REGION Network 6: Safety control condition 3
   // Do not allow any motion when the Object is in a collision with axes.
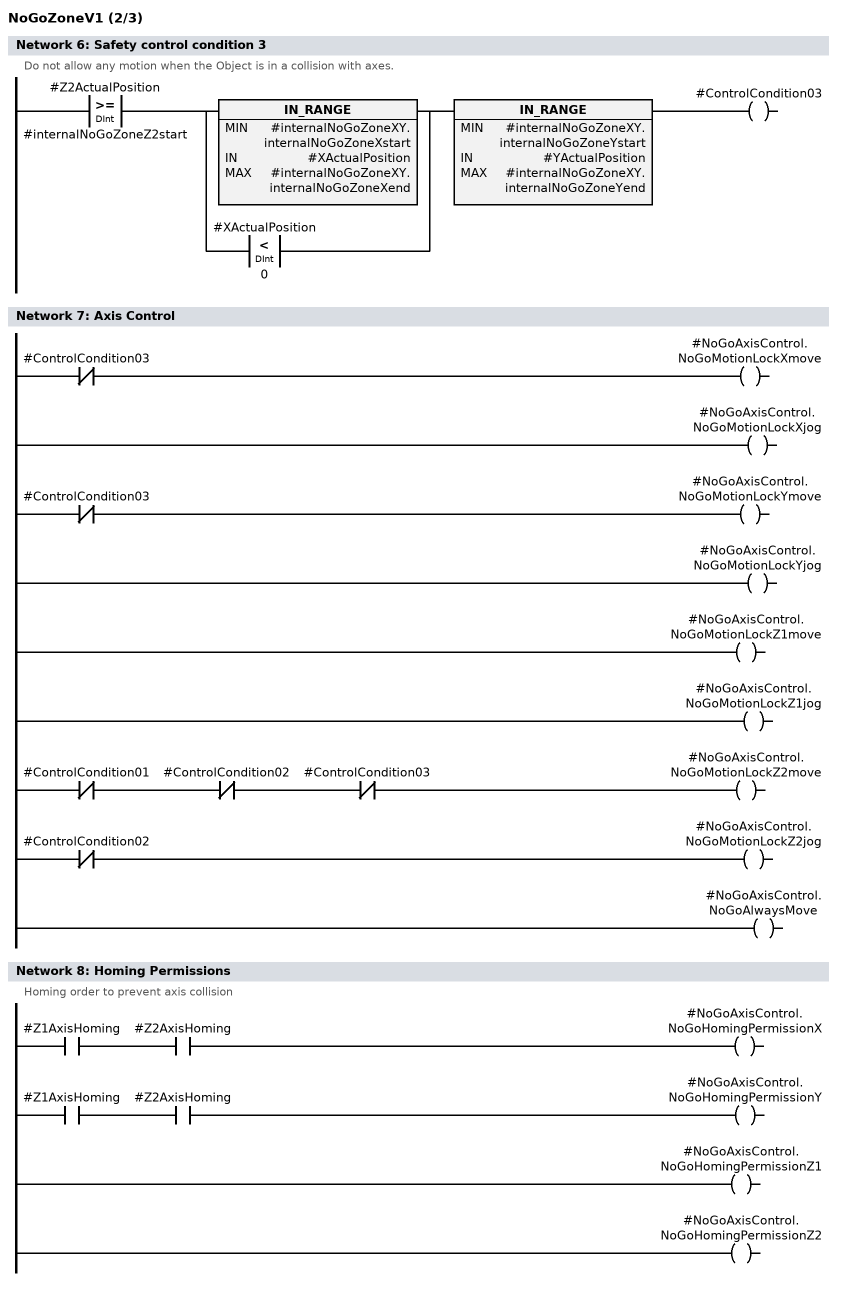
   RUNG wire#powerrail
      { S7_Templates := "SrcType := DInt" } GE_Contact(in1 := #Z2ActualPosition, in2 := #internalNoGoZoneZ2start)
      wire#w1
      { S7_Templates := "SrcType := DInt" } InRange(min := #internalNoGoZoneXY.internalNoGoZoneXstart, in := #XActualPosition, max := #internalNoGoZoneXY.internalNoGoZoneXend)
      wire#w2
      { S7_Templates := "SrcType := DInt" } InRange(min := #internalNoGoZoneXY.internalNoGoZoneYstart, in := #YActualPosition, max := #internalNoGoZoneXY.internalNoGoZoneYend)
      Coil( #ControlCondition03 )
   END_RUNG
   RUNG wire#w1
      { S7_Templates := "SrcType := DInt" } LT_Contact(in1 := #XActualPosition, in2 := 0)
   END_RUNG wire#w2
   // the same network as SCL:
   #ControlCondition03 := (#Z2ActualPosition >= #internalNoGoZoneZ2start) AND (((#internalNoGoZoneXY.internalNoGoZoneXstart <= #XActualPosition) AND (#XActualPosition <= #internalNoGoZoneXY.internalNoGoZoneXend)) OR (#XActualPosition < 0)) AND (#internalNoGoZoneXY.internalNoGoZoneYstart <= #YActualPosition) AND (#YActualPosition <= #internalNoGoZoneXY.internalNoGoZoneYend);
END_REGION

REGION Network 7: Axis Control
   RUNG wire#powerrail
      I_Contact( #ControlCondition03 )
      Coil( #NoGoAxisControl.NoGoMotionLockXmove )
   END_RUNG
   RUNG wire#powerrail
      Coil( #NoGoAxisControl.NoGoMotionLockXjog )
   END_RUNG
   RUNG wire#powerrail
      I_Contact( #ControlCondition03 )
      Coil( #NoGoAxisControl.NoGoMotionLockYmove )
   END_RUNG
   RUNG wire#powerrail
      Coil( #NoGoAxisControl.NoGoMotionLockYjog )
   END_RUNG
   RUNG wire#powerrail
      Coil( #NoGoAxisControl.NoGoMotionLockZ1move )
   END_RUNG
   RUNG wire#powerrail
      Coil( #NoGoAxisControl.NoGoMotionLockZ1jog )
   END_RUNG
   RUNG wire#powerrail
      I_Contact( #ControlCondition01 )
      I_Contact( #ControlCondition02 )
      I_Contact( #ControlCondition03 )
      Coil( #NoGoAxisControl.NoGoMotionLockZ2move )
   END_RUNG
   RUNG wire#powerrail
      I_Contact( #ControlCondition02 )
      Coil( #NoGoAxisControl.NoGoMotionLockZ2jog )
   END_RUNG
   RUNG wire#powerrail
      Coil( #NoGoAxisControl.NoGoAlwaysMove )
   END_RUNG
   // the same network as SCL:
   #NoGoAxisControl.NoGoMotionLockXmove := NOT #ControlCondition03;
   #NoGoAxisControl.NoGoMotionLockXjog := TRUE;
   #NoGoAxisControl.NoGoMotionLockYmove := NOT #ControlCondition03;
   #NoGoAxisControl.NoGoMotionLockYjog := TRUE;
   #NoGoAxisControl.NoGoMotionLockZ1move := TRUE;
   #NoGoAxisControl.NoGoMotionLockZ1jog := TRUE;
   #NoGoAxisControl.NoGoMotionLockZ2move := NOT #ControlCondition01 AND NOT #ControlCondition02 AND NOT #ControlCondition03;
   #NoGoAxisControl.NoGoMotionLockZ2jog := NOT #ControlCondition02;
   #NoGoAxisControl.NoGoAlwaysMove := TRUE;
END_REGION

REGION Network 8: Homing Permissions
   // Homing order to prevent axis collision
   RUNG wire#powerrail
      Contact( #Z1AxisHoming )
      Contact( #Z2AxisHoming )
      Coil( #NoGoAxisControl.NoGoHomingPermissionX )
   END_RUNG
   RUNG wire#powerrail
      Contact( #Z1AxisHoming )
      Contact( #Z2AxisHoming )
      Coil( #NoGoAxisControl.NoGoHomingPermissionY )
   END_RUNG
   RUNG wire#powerrail
      Coil( #NoGoAxisControl.NoGoHomingPermissionZ1 )
   END_RUNG
   RUNG wire#powerrail
      Coil( #NoGoAxisControl.NoGoHomingPermissionZ2 )
   END_RUNG
   // the same network as SCL:
   #NoGoAxisControl.NoGoHomingPermissionX := #Z1AxisHoming AND #Z2AxisHoming;
   #NoGoAxisControl.NoGoHomingPermissionY := #Z1AxisHoming AND #Z2AxisHoming;
   #NoGoAxisControl.NoGoHomingPermissionZ1 := TRUE;
   #NoGoAxisControl.NoGoHomingPermissionZ2 := TRUE;
END_REGION

REGION Network 9: Status
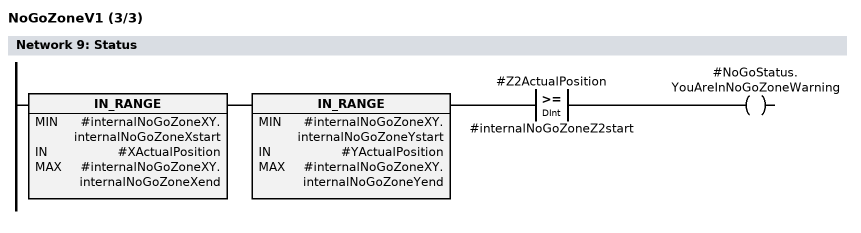
   RUNG wire#powerrail
      { S7_Templates := "SrcType := DInt" } InRange(min := #internalNoGoZoneXY.internalNoGoZoneXstart, in := #XActualPosition, max := #internalNoGoZoneXY.internalNoGoZoneXend)
      { S7_Templates := "SrcType := DInt" } InRange(min := #internalNoGoZoneXY.internalNoGoZoneYstart, in := #YActualPosition, max := #internalNoGoZoneXY.internalNoGoZoneYend)
      { S7_Templates := "SrcType := DInt" } GE_Contact(in1 := #Z2ActualPosition, in2 := #internalNoGoZoneZ2start)
      Coil( #NoGoStatus.YouAreInNoGoZoneWarning )
   END_RUNG
   // the same network as SCL:
   #NoGoStatus.YouAreInNoGoZoneWarning := (#internalNoGoZoneXY.internalNoGoZoneXstart <= #XActualPosition) AND (#XActualPosition <= #internalNoGoZoneXY.internalNoGoZoneXend) AND (#internalNoGoZoneXY.internalNoGoZoneYstart <= #YActualPosition) AND (#YActualPosition <= #internalNoGoZoneXY.internalNoGoZoneYend) AND (#Z2ActualPosition >= #internalNoGoZoneZ2start);
END_REGION
END_FUNCTION_BLOCK

FUNCTION "Reset Error" : Void   // FC15, LAD
{ S7_Optimized_Access := 'TRUE' }
AUTHOR : HenriP
VERSION : 0.1
   VAR_INPUT
      FestoAxisFault : Bool;
   END_VAR
   VAR_IN_OUT
      ResetCommand : Bool;
      FestoReset : Bool;
   END_VAR
BEGIN

REGION Network 1: Send Reset Command Flip Flop logic on Command
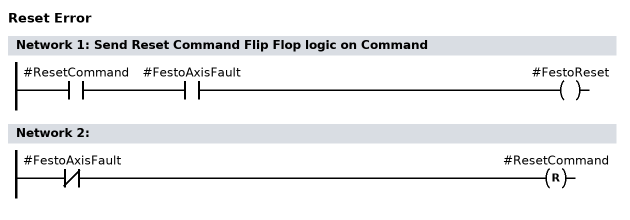
   RUNG wire#powerrail
      Contact( #ResetCommand )
      Contact( #FestoAxisFault )
      Coil( #FestoReset )
   END_RUNG
   // the same network as SCL:
   #FestoReset := #ResetCommand AND #FestoAxisFault;
END_REGION

REGION Network 2
   RUNG wire#powerrail
      I_Contact( #FestoAxisFault )
      R_Coil( #ResetCommand )
   END_RUNG
   // the same network as SCL:
   IF NOT #FestoAxisFault THEN #ResetCommand := FALSE; END_IF;
END_REGION
END_FUNCTION

ORGANIZATION_BLOCK "Startup"   // OB100, LAD, Startup
TITLE = "Complete Restart"
{ S7_Optimized_Access := 'TRUE' }
AUTHOR : HenriP
VERSION : 0.1
   VAR_INPUT
      LostRetentive : Bool;   // True if retentive data are lost
      LostRTC : Bool;   // True if date and time are lost
   END_VAR
   VAR_TEMP
      InitCall : Bool;
   END_VAR
BEGIN

REGION Network 1: Startup
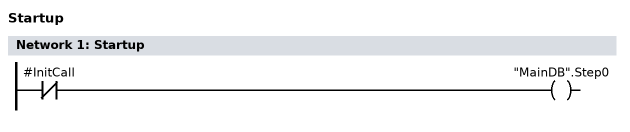
   RUNG wire#powerrail
      I_Contact( #InitCall )
      Coil( "MainDB".Step0 )
   END_RUNG
   // the same network as SCL:
   "MainDB".Step0 := NOT #InitCall;
END_REGION
END_ORGANIZATION_BLOCK

ORGANIZATION_BLOCK "Status Monitor"   // OB127, LAD, ProgramCycle
TITLE = Main Control block
{ S7_Optimized_Access := 'TRUE' }
AUTHOR : HenriP
VERSION : 0.1
   VAR_INPUT
      Initial_Call : Bool;   // Initial call of this OB
      Remanence : Bool;   // =True, if remanent data are available
   END_VAR
   VAR_TEMP
      ClearError : Bool;
   END_VAR
   VAR_TEMP   // added for the SCL form of the ladder/FBD networks
      _w1 : Bool;
   END_VAR
BEGIN

REGION Network 1: Monitor
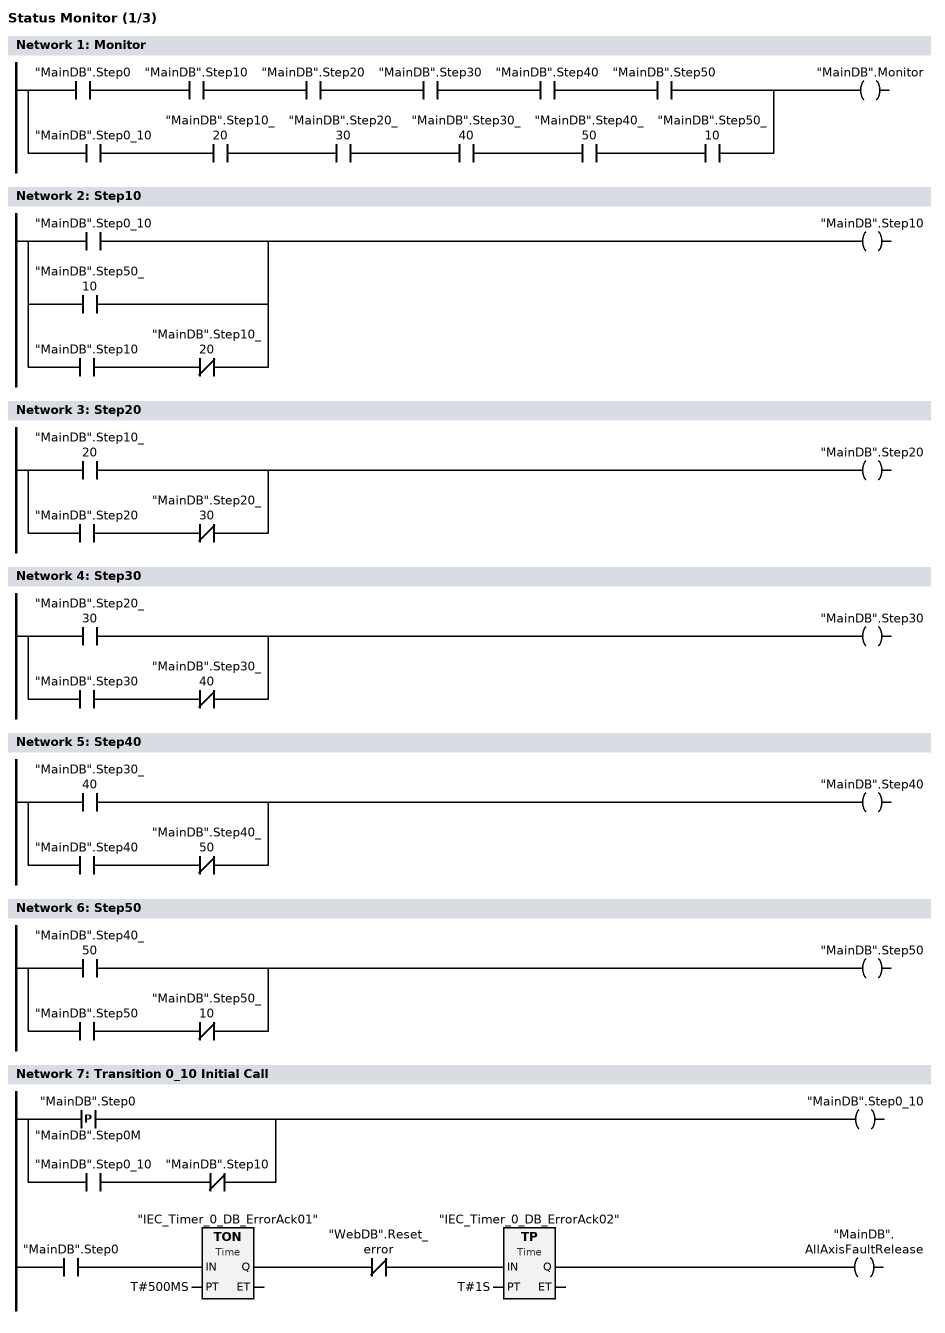
   RUNG wire#powerrail
      Contact( "MainDB".Step0 )
      Contact( "MainDB".Step10 )
      Contact( "MainDB".Step20 )
      Contact( "MainDB".Step30 )
      Contact( "MainDB".Step40 )
      Contact( "MainDB".Step50 )
      wire#w1
      Coil( "MainDB".Monitor )
   END_RUNG
   RUNG wire#powerrail
      Contact( "MainDB".Step0_10 )
      Contact( "MainDB".Step10_20 )
      Contact( "MainDB".Step20_30 )
      Contact( "MainDB".Step30_40 )
      Contact( "MainDB".Step40_50 )
      Contact( "MainDB".Step50_10 )
   END_RUNG wire#w1
   // the same network as SCL:
   "MainDB".Monitor := ("MainDB".Step0 AND "MainDB".Step10 AND "MainDB".Step20 AND "MainDB".Step30 AND "MainDB".Step40 AND "MainDB".Step50) OR ("MainDB".Step0_10 AND "MainDB".Step10_20 AND "MainDB".Step20_30 AND "MainDB".Step30_40 AND "MainDB".Step40_50 AND "MainDB".Step50_10);
END_REGION

REGION Network 2: Step10
   RUNG wire#powerrail
      Contact( "MainDB".Step0_10 )
      wire#w1
      Coil( "MainDB".Step10 )
   END_RUNG
   RUNG wire#powerrail
      Contact( "MainDB".Step50_10 )
   END_RUNG wire#w1
   RUNG wire#powerrail
      Contact( "MainDB".Step10 )
      I_Contact( "MainDB".Step10_20 )
   END_RUNG wire#w1
   // the same network as SCL:
   "MainDB".Step10 := "MainDB".Step0_10 OR "MainDB".Step50_10 OR ("MainDB".Step10 AND NOT "MainDB".Step10_20);
END_REGION

REGION Network 3: Step20
   RUNG wire#powerrail
      Contact( "MainDB".Step10_20 )
      wire#w1
      Coil( "MainDB".Step20 )
   END_RUNG
   RUNG wire#powerrail
      Contact( "MainDB".Step20 )
      I_Contact( "MainDB".Step20_30 )
   END_RUNG wire#w1
   // the same network as SCL:
   "MainDB".Step20 := "MainDB".Step10_20 OR ("MainDB".Step20 AND NOT "MainDB".Step20_30);
END_REGION

REGION Network 4: Step30
   RUNG wire#powerrail
      Contact( "MainDB".Step20_30 )
      wire#w1
      Coil( "MainDB".Step30 )
   END_RUNG
   RUNG wire#powerrail
      Contact( "MainDB".Step30 )
      I_Contact( "MainDB".Step30_40 )
   END_RUNG wire#w1
   // the same network as SCL:
   "MainDB".Step30 := "MainDB".Step20_30 OR ("MainDB".Step30 AND NOT "MainDB".Step30_40);
END_REGION

REGION Network 5: Step40
   RUNG wire#powerrail
      Contact( "MainDB".Step30_40 )
      wire#w1
      Coil( "MainDB".Step40 )
   END_RUNG
   RUNG wire#powerrail
      Contact( "MainDB".Step40 )
      I_Contact( "MainDB".Step40_50 )
   END_RUNG wire#w1
   // the same network as SCL:
   "MainDB".Step40 := "MainDB".Step30_40 OR ("MainDB".Step40 AND NOT "MainDB".Step40_50);
END_REGION

REGION Network 6: Step50
   RUNG wire#powerrail
      Contact( "MainDB".Step40_50 )
      wire#w1
      Coil( "MainDB".Step50 )
   END_RUNG
   RUNG wire#powerrail
      Contact( "MainDB".Step50 )
      I_Contact( "MainDB".Step50_10 )
   END_RUNG wire#w1
   // the same network as SCL:
   "MainDB".Step50 := "MainDB".Step40_50 OR ("MainDB".Step50 AND NOT "MainDB".Step50_10);
END_REGION

REGION Network 7: Transition 0_10 Initial Call
   RUNG wire#powerrail
      P_Contact(operand := "MainDB".Step0, bit := "MainDB".Step0M)
      wire#w1
      Coil( "MainDB".Step0_10 )
   END_RUNG
   RUNG wire#powerrail
      Contact( "MainDB".Step0_10 )
      I_Contact( "MainDB".Step10 )
   END_RUNG wire#w1
   RUNG wire#powerrail
      Contact( "MainDB".Step0 )
      { S7_Templates := "time_type := Time" } "IEC_Timer_0_DB_ErrorAck01".TON(pt := T#500MS, et =>)
      I_Contact( "WebDB".Reset_error )
      { S7_Templates := "time_type := Time" } "IEC_Timer_0_DB_ErrorAck02".TP(pt := T#1S, et =>)
      Coil( "MainDB".AllAxisFaultRelease )
   END_RUNG
   // the same network as SCL:
   #_w1 := "MainDB".Step0 AND NOT "MainDB".Step0M;   // rising edge of "MainDB".Step0
   "MainDB".Step0M := "MainDB".Step0;
   "MainDB".Step0_10 := #_w1 OR ("MainDB".Step0_10 AND NOT "MainDB".Step10);
   "IEC_Timer_0_DB_ErrorAck01".TON(IN := "MainDB".Step0, PT := T#500MS);
   "IEC_Timer_0_DB_ErrorAck02".TP(IN := "IEC_Timer_0_DB_ErrorAck01".Q AND NOT "WebDB".Reset_error, PT := T#1S);
   "MainDB".AllAxisFaultRelease := "IEC_Timer_0_DB_ErrorAck02".Q;
END_REGION

REGION Network 8: Transition10-20 Check PLC Operating State -> Wait Ready
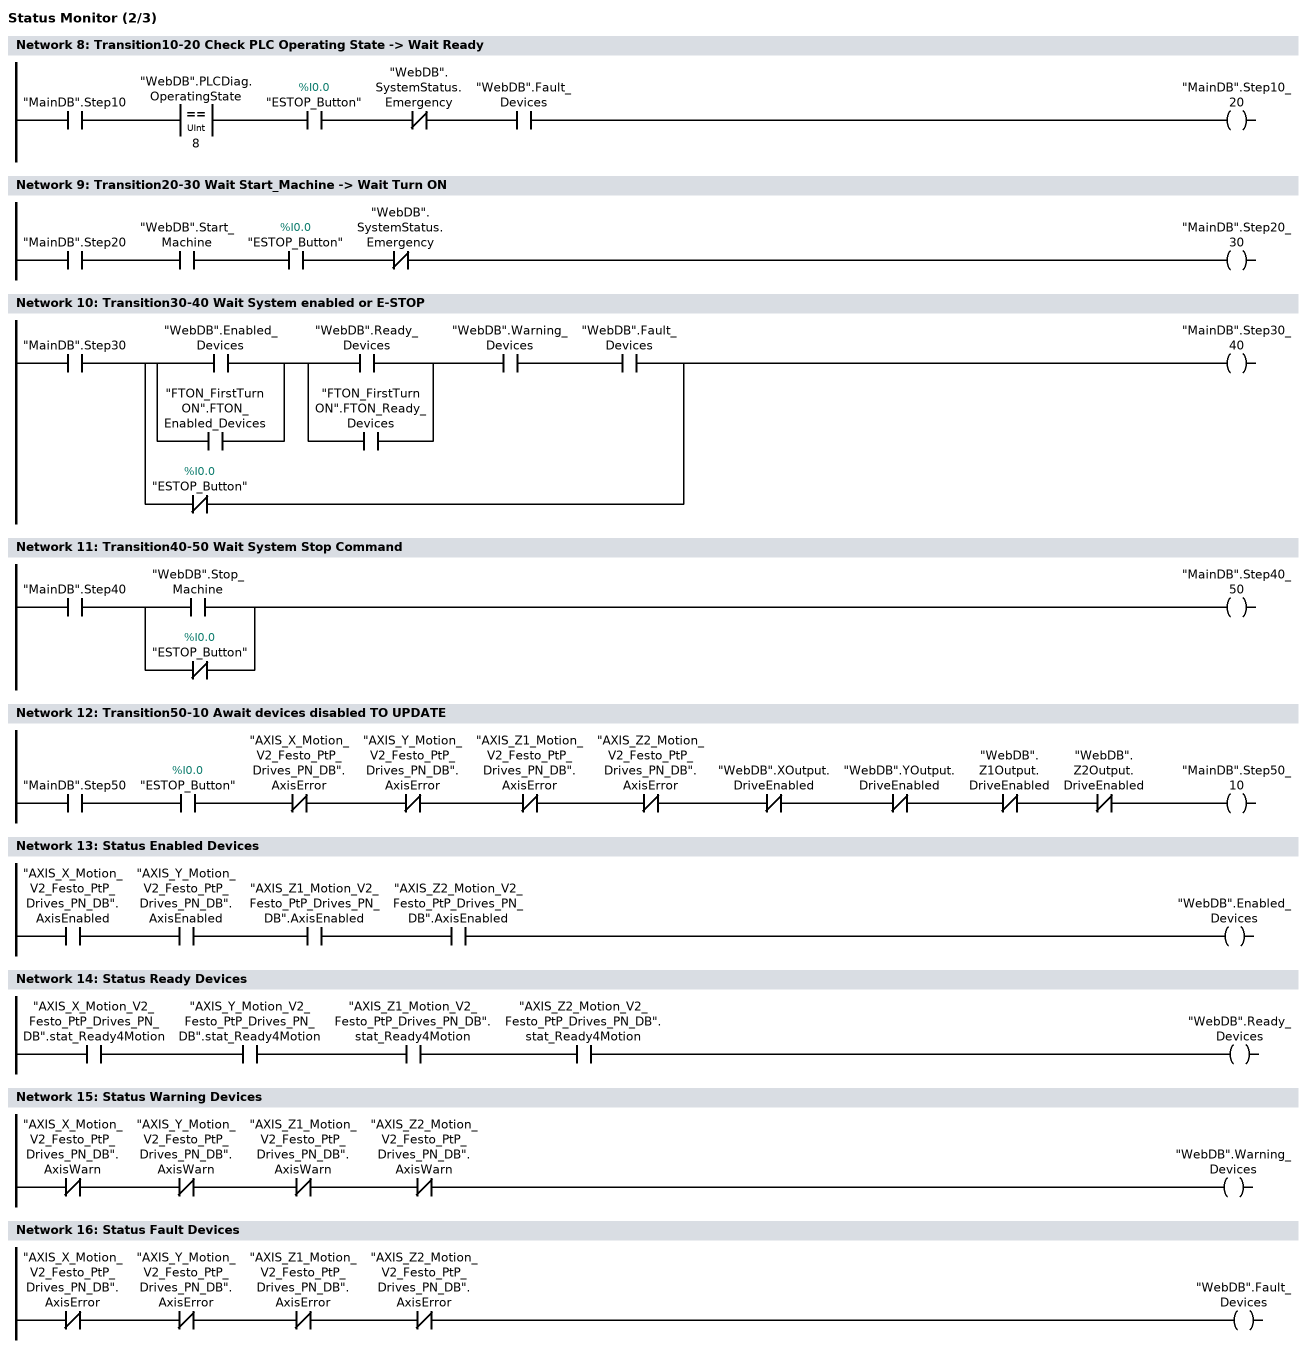
   RUNG wire#powerrail
      Contact( "MainDB".Step10 )
      { S7_Templates := "SrcType := UInt" } EQ_Contact(in1 := "WebDB".PLCDiag.OperatingState, in2 := 8)
      Contact( "ESTOP_Button" )
      I_Contact( "WebDB".SystemStatus.Emergency )
      Contact( "WebDB".Fault_Devices )
      Coil( "MainDB".Step10_20 )
   END_RUNG
   // the same network as SCL:
   "MainDB".Step10_20 := "MainDB".Step10 AND ("WebDB".PLCDiag.OperatingState = 8) AND "ESTOP_Button" AND NOT "WebDB".SystemStatus.Emergency AND "WebDB".Fault_Devices;
END_REGION

REGION Network 9: Transition20-30 Wait Start_Machine -> Wait Turn ON
   RUNG wire#powerrail
      Contact( "MainDB".Step20 )
      Contact( "WebDB".Start_Machine )
      Contact( "ESTOP_Button" )
      I_Contact( "WebDB".SystemStatus.Emergency )
      Coil( "MainDB".Step20_30 )
   END_RUNG
   // the same network as SCL:
   "MainDB".Step20_30 := "MainDB".Step20 AND "WebDB".Start_Machine AND "ESTOP_Button" AND NOT "WebDB".SystemStatus.Emergency;
END_REGION

REGION Network 10: Transition30-40 Wait System enabled or E-STOP
   RUNG wire#powerrail
      Contact( "MainDB".Step30 )
      wire#w1
      Contact( "WebDB".Enabled_Devices )
      wire#w2
      Contact( "WebDB".Ready_Devices )
      wire#w3
      Contact( "WebDB".Warning_Devices )
      Contact( "WebDB".Fault_Devices )
      wire#w4
      Coil( "MainDB".Step30_40 )
   END_RUNG
   RUNG wire#w1
      Contact( "FTON_FirstTurnON".FTON_Enabled_Devices )
   END_RUNG wire#w2
   RUNG wire#w2
      Contact( "FTON_FirstTurnON".FTON_Ready_Devices )
   END_RUNG wire#w3
   RUNG wire#w1
      I_Contact( "ESTOP_Button" )
   END_RUNG wire#w4
   // the same network as SCL:
   "MainDB".Step30_40 := "MainDB".Step30 AND ((("WebDB".Enabled_Devices OR "FTON_FirstTurnON".FTON_Enabled_Devices) AND ("WebDB".Ready_Devices OR "FTON_FirstTurnON".FTON_Ready_Devices) AND "WebDB".Warning_Devices AND "WebDB".Fault_Devices) OR NOT "ESTOP_Button");
END_REGION

REGION Network 11: Transition40-50 Wait System Stop Command
   RUNG wire#powerrail
      Contact( "MainDB".Step40 )
      wire#w1
      Contact( "WebDB".Stop_Machine )
      wire#w2
      Coil( "MainDB".Step40_50 )
   END_RUNG
   RUNG wire#w1
      I_Contact( "ESTOP_Button" )
   END_RUNG wire#w2
   // the same network as SCL:
   "MainDB".Step40_50 := "MainDB".Step40 AND ("WebDB".Stop_Machine OR NOT "ESTOP_Button");
END_REGION

REGION Network 12: Transition50-10 Await devices disabled TO UPDATE
   RUNG wire#powerrail
      Contact( "MainDB".Step50 )
      Contact( "ESTOP_Button" )
      I_Contact( "AXIS_X_Motion_V2_Festo_PtP_Drives_PN_DB".AxisError )
      I_Contact( "AXIS_Y_Motion_V2_Festo_PtP_Drives_PN_DB".AxisError )
      I_Contact( "AXIS_Z1_Motion_V2_Festo_PtP_Drives_PN_DB".AxisError )
      I_Contact( "AXIS_Z2_Motion_V2_Festo_PtP_Drives_PN_DB".AxisError )
      I_Contact( "WebDB".XOutput.DriveEnabled )
      I_Contact( "WebDB".YOutput.DriveEnabled )
      I_Contact( "WebDB".Z1Output.DriveEnabled )
      I_Contact( "WebDB".Z2Output.DriveEnabled )
      Coil( "MainDB".Step50_10 )
   END_RUNG
   // the same network as SCL:
   "MainDB".Step50_10 := "MainDB".Step50 AND "ESTOP_Button" AND NOT "AXIS_X_Motion_V2_Festo_PtP_Drives_PN_DB".AxisError AND NOT "AXIS_Y_Motion_V2_Festo_PtP_Drives_PN_DB".AxisError AND NOT "AXIS_Z1_Motion_V2_Festo_PtP_Drives_PN_DB".AxisError AND NOT "AXIS_Z2_Motion_V2_Festo_PtP_Drives_PN_DB".AxisError AND NOT "WebDB".XOutput.DriveEnabled AND NOT "WebDB".YOutput.DriveEnabled AND NOT "WebDB".Z1Output.DriveEnabled AND NOT "WebDB".Z2Output.DriveEnabled;
END_REGION

REGION Network 13: Status Enabled Devices
   RUNG wire#powerrail
      Contact( "AXIS_X_Motion_V2_Festo_PtP_Drives_PN_DB".AxisEnabled )
      Contact( "AXIS_Y_Motion_V2_Festo_PtP_Drives_PN_DB".AxisEnabled )
      Contact( "AXIS_Z1_Motion_V2_Festo_PtP_Drives_PN_DB".AxisEnabled )
      Contact( "AXIS_Z2_Motion_V2_Festo_PtP_Drives_PN_DB".AxisEnabled )
      Coil( "WebDB".Enabled_Devices )
   END_RUNG
   // the same network as SCL:
   "WebDB".Enabled_Devices := "AXIS_X_Motion_V2_Festo_PtP_Drives_PN_DB".AxisEnabled AND "AXIS_Y_Motion_V2_Festo_PtP_Drives_PN_DB".AxisEnabled AND "AXIS_Z1_Motion_V2_Festo_PtP_Drives_PN_DB".AxisEnabled AND "AXIS_Z2_Motion_V2_Festo_PtP_Drives_PN_DB".AxisEnabled;
END_REGION

REGION Network 14: Status Ready Devices
   RUNG wire#powerrail
      Contact( "AXIS_X_Motion_V2_Festo_PtP_Drives_PN_DB".stat_Ready4Motion )
      Contact( "AXIS_Y_Motion_V2_Festo_PtP_Drives_PN_DB".stat_Ready4Motion )
      Contact( "AXIS_Z1_Motion_V2_Festo_PtP_Drives_PN_DB".stat_Ready4Motion )
      Contact( "AXIS_Z2_Motion_V2_Festo_PtP_Drives_PN_DB".stat_Ready4Motion )
      Coil( "WebDB".Ready_Devices )
   END_RUNG
   // the same network as SCL:
   "WebDB".Ready_Devices := "AXIS_X_Motion_V2_Festo_PtP_Drives_PN_DB".stat_Ready4Motion AND "AXIS_Y_Motion_V2_Festo_PtP_Drives_PN_DB".stat_Ready4Motion AND "AXIS_Z1_Motion_V2_Festo_PtP_Drives_PN_DB".stat_Ready4Motion AND "AXIS_Z2_Motion_V2_Festo_PtP_Drives_PN_DB".stat_Ready4Motion;
END_REGION

REGION Network 15: Status Warning Devices
   RUNG wire#powerrail
      I_Contact( "AXIS_X_Motion_V2_Festo_PtP_Drives_PN_DB".AxisWarn )
      I_Contact( "AXIS_Y_Motion_V2_Festo_PtP_Drives_PN_DB".AxisWarn )
      I_Contact( "AXIS_Z1_Motion_V2_Festo_PtP_Drives_PN_DB".AxisWarn )
      I_Contact( "AXIS_Z2_Motion_V2_Festo_PtP_Drives_PN_DB".AxisWarn )
      Coil( "WebDB".Warning_Devices )
   END_RUNG
   // the same network as SCL:
   "WebDB".Warning_Devices := NOT "AXIS_X_Motion_V2_Festo_PtP_Drives_PN_DB".AxisWarn AND NOT "AXIS_Y_Motion_V2_Festo_PtP_Drives_PN_DB".AxisWarn AND NOT "AXIS_Z1_Motion_V2_Festo_PtP_Drives_PN_DB".AxisWarn AND NOT "AXIS_Z2_Motion_V2_Festo_PtP_Drives_PN_DB".AxisWarn;
END_REGION

REGION Network 16: Status Fault Devices
   RUNG wire#powerrail
      I_Contact( "AXIS_X_Motion_V2_Festo_PtP_Drives_PN_DB".AxisError )
      I_Contact( "AXIS_Y_Motion_V2_Festo_PtP_Drives_PN_DB".AxisError )
      I_Contact( "AXIS_Z1_Motion_V2_Festo_PtP_Drives_PN_DB".AxisError )
      I_Contact( "AXIS_Z2_Motion_V2_Festo_PtP_Drives_PN_DB".AxisError )
      Coil( "WebDB".Fault_Devices )
   END_RUNG
   // the same network as SCL:
   "WebDB".Fault_Devices := NOT "AXIS_X_Motion_V2_Festo_PtP_Drives_PN_DB".AxisError AND NOT "AXIS_Y_Motion_V2_Festo_PtP_Drives_PN_DB".AxisError AND NOT "AXIS_Z1_Motion_V2_Festo_PtP_Drives_PN_DB".AxisError AND NOT "AXIS_Z2_Motion_V2_Festo_PtP_Drives_PN_DB".AxisError;
END_REGION

REGION Network 17: Emergency button is active
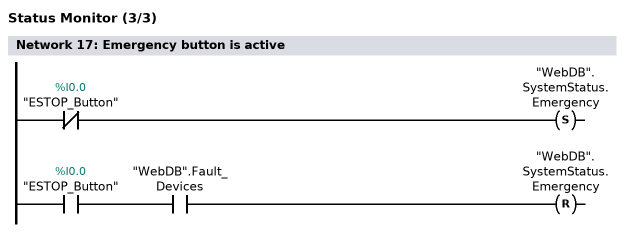
   RUNG wire#powerrail
      I_Contact( "ESTOP_Button" )
      S_Coil( "WebDB".SystemStatus.Emergency )
   END_RUNG
   RUNG wire#powerrail
      Contact( "ESTOP_Button" )
      Contact( "WebDB".Fault_Devices )
      R_Coil( "WebDB".SystemStatus.Emergency )
   END_RUNG
   // the same network as SCL:
   IF NOT "ESTOP_Button" THEN "WebDB".SystemStatus.Emergency := TRUE; END_IF;
   IF "ESTOP_Button" AND "WebDB".Fault_Devices THEN "WebDB".SystemStatus.Emergency := FALSE; END_IF;
END_REGION
END_ORGANIZATION_BLOCK

ORGANIZATION_BLOCK "Work"   // OB123, LAD, ProgramCycle
TITLE = "Main Program Sweep (Cycle)"
{ S7_Optimized_Access := 'TRUE' }
VERSION : 0.1
   VAR_INPUT
      Initial_Call : Bool;   // Initial call of this OB
      Remanence : Bool;   // =True, if remanent data are available
   END_VAR
BEGIN

REGION Network 1: Active machine
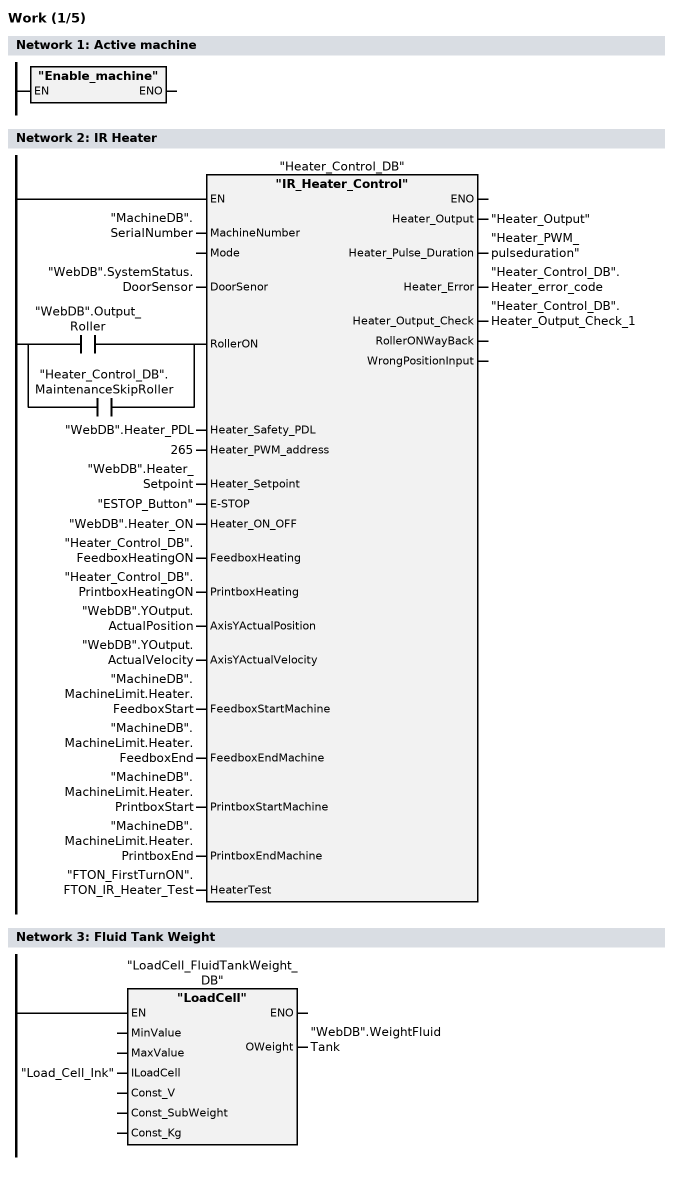
   RUNG wire#powerrail
      "Enable_machine"()
   END_RUNG
   // the same network as SCL:
   "Enable_machine"();
END_REGION

REGION Network 2: IR Heater
   RUNG wire#powerrail
      "Heater_Control_DB"(RollerON := wire#w1, MachineNumber := "MachineDB".SerialNumber, Mode :=, DoorSenor := "WebDB".SystemStatus.DoorSensor, Heater_Safety_PDL := "WebDB".Heater_PDL, Heater_PWM_address := 265, Heater_Setpoint := "WebDB".Heater_Setpoint, "E-STOP" := "ESTOP_Button", Heater_ON_OFF := "WebDB".Heater_ON, FeedboxHeating := "Heater_Control_DB".FeedboxHeatingON, PrintboxHeating := "Heater_Control_DB".PrintboxHeatingON, AxisYActualPosition := "WebDB".YOutput.ActualPosition, AxisYActualVelocity := "WebDB".YOutput.ActualVelocity, FeedboxStartMachine := "MachineDB".MachineLimit.Heater.FeedboxStart, FeedboxEndMachine := "MachineDB".MachineLimit.Heater.FeedboxEnd, PrintboxStartMachine := "MachineDB".MachineLimit.Heater.PrintboxStart, PrintboxEndMachine := "MachineDB".MachineLimit.Heater.PrintboxEnd, HeaterTest := "FTON_FirstTurnON".FTON_IR_Heater_Test, Heater_Output => "Heater_Output", Heater_Pulse_Duration => "Heater_PWM_pulseduration", Heater_Error => "Heater_Control_DB".Heater_error_code, Heater_Output_Check => "Heater_Control_DB".Heater_Output_Check_1, RollerONWayBack =>, WrongPositionInput =>)
   END_RUNG
   RUNG wire#powerrail
      Contact( "WebDB".Output_Roller )
   END_RUNG wire#w1
   RUNG wire#powerrail
      Contact( "Heater_Control_DB".MaintenanceSkipRoller )
   END_RUNG wire#w1
   // the same network as SCL:
   "Heater_Control_DB"(MachineNumber := "MachineDB".SerialNumber,   // "IR_Heater_Control"
                       DoorSenor := "WebDB".SystemStatus.DoorSensor,
                       RollerON := "WebDB".Output_Roller OR "Heater_Control_DB".MaintenanceSkipRoller,
                       Heater_Safety_PDL := "WebDB".Heater_PDL,
                       Heater_PWM_address := 265,
                       Heater_Setpoint := "WebDB".Heater_Setpoint,
                       "E-STOP" := "ESTOP_Button",
                       Heater_ON_OFF := "WebDB".Heater_ON,
                       FeedboxHeating := "Heater_Control_DB".FeedboxHeatingON,
                       PrintboxHeating := "Heater_Control_DB".PrintboxHeatingON,
                       AxisYActualPosition := "WebDB".YOutput.ActualPosition,
                       AxisYActualVelocity := "WebDB".YOutput.ActualVelocity,
                       FeedboxStartMachine := "MachineDB".MachineLimit.Heater.FeedboxStart,
                       FeedboxEndMachine := "MachineDB".MachineLimit.Heater.FeedboxEnd,
                       PrintboxStartMachine := "MachineDB".MachineLimit.Heater.PrintboxStart,
                       PrintboxEndMachine := "MachineDB".MachineLimit.Heater.PrintboxEnd,
                       HeaterTest := "FTON_FirstTurnON".FTON_IR_Heater_Test,
                       Heater_Output => "Heater_Output",
                       Heater_Pulse_Duration => "Heater_PWM_pulseduration",
                       Heater_Error => "Heater_Control_DB".Heater_error_code,
                       Heater_Output_Check => "Heater_Control_DB".Heater_Output_Check_1);
END_REGION

REGION Network 3: Fluid Tank Weight
   RUNG wire#powerrail
      "LoadCell_FluidTankWeight_DB"(MinValue :=, MaxValue :=, ILoadCell := "Load_Cell_Ink", Const_V :=, Const_SubWeight :=, Const_Kg :=, OWeight => "WebDB".WeightFluidTank)
   END_RUNG
   // the same network as SCL:
   "LoadCell_FluidTankWeight_DB"(ILoadCell := "Load_Cell_Ink", OWeight => "WebDB".WeightFluidTank);   // "LoadCell"
END_REGION

REGION Network 4: Fluid Waste Weight
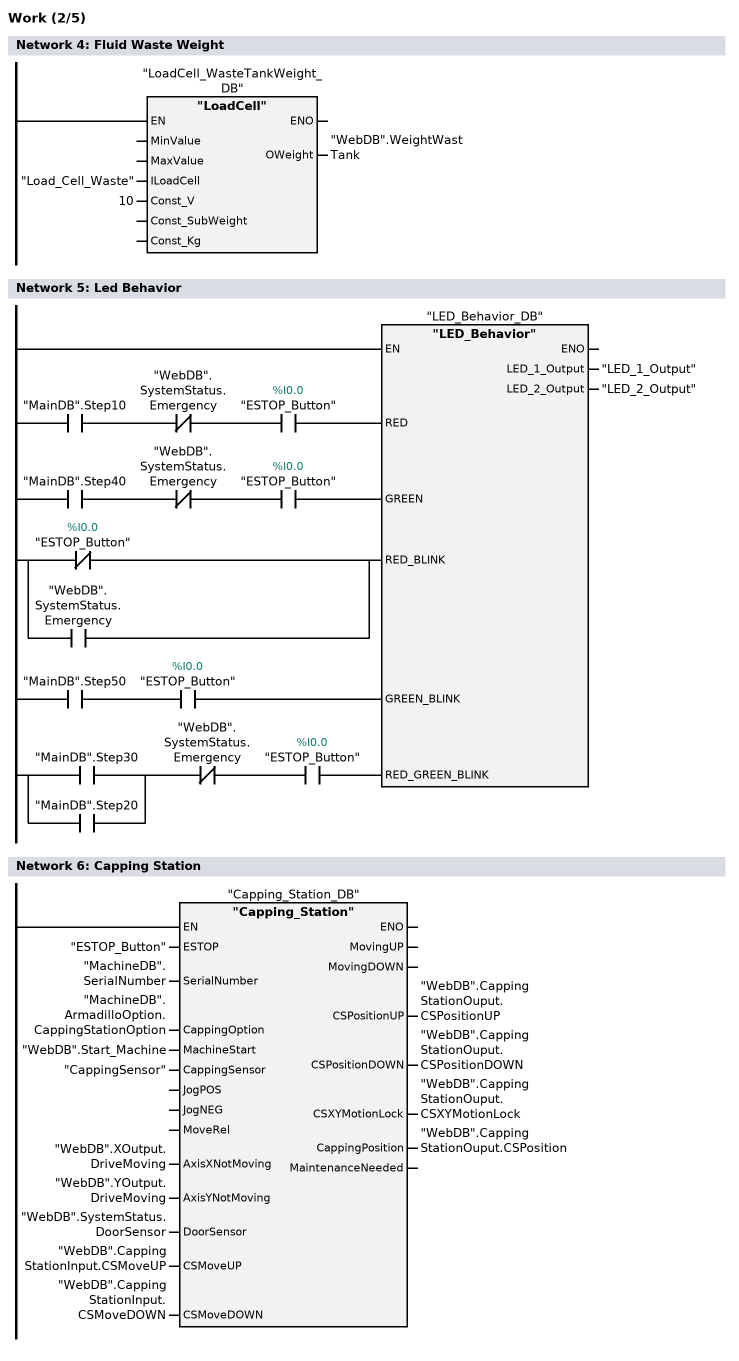
   RUNG wire#powerrail
      "LoadCell_WasteTankWeight_DB"(MinValue :=, MaxValue :=, ILoadCell := "Load_Cell_Waste", Const_V := 10, Const_SubWeight :=, Const_Kg :=, OWeight => "WebDB".WeightWastTank)
   END_RUNG
   // the same network as SCL:
   "LoadCell_WasteTankWeight_DB"(ILoadCell := "Load_Cell_Waste",   // "LoadCell"
                           Const_V := 10,
                           OWeight => "WebDB".WeightWastTank);
END_REGION

REGION Network 5: Led Behavior
   RUNG wire#powerrail
      "LED_Behavior_DB"(RED := wire#w1, GREEN := wire#w2, RED_BLINK := wire#w3, GREEN_BLINK := wire#w4, RED_GREEN_BLINK := wire#w6, LED_1_Output => "LED_1_Output", LED_2_Output => "LED_2_Output")
   END_RUNG
   RUNG wire#powerrail
      Contact( "MainDB".Step10 )
      I_Contact( "WebDB".SystemStatus.Emergency )
      Contact( "ESTOP_Button" )
   END_RUNG wire#w1
   RUNG wire#powerrail
      Contact( "MainDB".Step40 )
      I_Contact( "WebDB".SystemStatus.Emergency )
      Contact( "ESTOP_Button" )
   END_RUNG wire#w2
   RUNG wire#powerrail
      I_Contact( "ESTOP_Button" )
   END_RUNG wire#w3
   RUNG wire#powerrail
      Contact( "WebDB".SystemStatus.Emergency )
   END_RUNG wire#w3
   RUNG wire#powerrail
      Contact( "MainDB".Step50 )
      Contact( "ESTOP_Button" )
   END_RUNG wire#w4
   RUNG wire#powerrail
      Contact( "MainDB".Step30 )
      wire#w5
      I_Contact( "WebDB".SystemStatus.Emergency )
      Contact( "ESTOP_Button" )
   END_RUNG wire#w6
   RUNG wire#powerrail
      Contact( "MainDB".Step20 )
   END_RUNG wire#w5
   // the same network as SCL:
   "LED_Behavior_DB"(RED := "MainDB".Step10 AND NOT "WebDB".SystemStatus.Emergency AND "ESTOP_Button",   // "LED_Behavior"
                     GREEN := "MainDB".Step40 AND NOT "WebDB".SystemStatus.Emergency AND "ESTOP_Button",
                     RED_BLINK := NOT "ESTOP_Button" OR "WebDB".SystemStatus.Emergency,
                     GREEN_BLINK := "MainDB".Step50 AND "ESTOP_Button",
                     RED_GREEN_BLINK := ("MainDB".Step30 OR "MainDB".Step20) AND NOT "WebDB".SystemStatus.Emergency AND "ESTOP_Button",
                     LED_1_Output => "LED_1_Output",
                     LED_2_Output => "LED_2_Output");
END_REGION

REGION Network 6: Capping Station
   RUNG wire#powerrail
      "Capping_Station_DB"(ESTOP := "ESTOP_Button", SerialNumber := "MachineDB".SerialNumber, CappingOption := "MachineDB".ArmadilloOption.CappingStationOption, MachineStart := "WebDB".Start_Machine, CappingSensor := "CappingSensor", JogPOS :=, JogNEG :=, MoveRel :=, AxisXNotMoving := "WebDB".XOutput.DriveMoving, AxisYNotMoving := "WebDB".YOutput.DriveMoving, DoorSensor := "WebDB".SystemStatus.DoorSensor, CSMoveUP := "WebDB".CappingStationInput.CSMoveUP, CSMoveDOWN := "WebDB".CappingStationInput.CSMoveDOWN, MovingUP =>, MovingDOWN =>, CSPositionUP => "WebDB".CappingStationOuput.CSPositionUP, CSPositionDOWN => "WebDB".CappingStationOuput.CSPositionDOWN, CSXYMotionLock => "WebDB".CappingStationOuput.CSXYMotionLock, CappingPosition => "WebDB".CappingStationOuput.CSPosition, MaintenanceNeeded =>)
   END_RUNG
   // the same network as SCL:
   "Capping_Station_DB"(ESTOP := "ESTOP_Button",   // "Capping_Station"
                        SerialNumber := "MachineDB".SerialNumber,
                        CappingOption := "MachineDB".ArmadilloOption.CappingStationOption,
                        MachineStart := "WebDB".Start_Machine,
                        CappingSensor := "CappingSensor",
                        AxisXNotMoving := "WebDB".XOutput.DriveMoving,
                        AxisYNotMoving := "WebDB".YOutput.DriveMoving,
                        DoorSensor := "WebDB".SystemStatus.DoorSensor,
                        CSMoveUP := "WebDB".CappingStationInput.CSMoveUP,
                        CSMoveDOWN := "WebDB".CappingStationInput.CSMoveDOWN,
                        CSPositionUP => "WebDB".CappingStationOuput.CSPositionUP,
                        CSPositionDOWN => "WebDB".CappingStationOuput.CSPositionDOWN,
                        CSXYMotionLock => "WebDB".CappingStationOuput.CSXYMotionLock,
                        CappingPosition => "WebDB".CappingStationOuput.CSPosition);
END_REGION

REGION Network 7: Initial Test Sequence
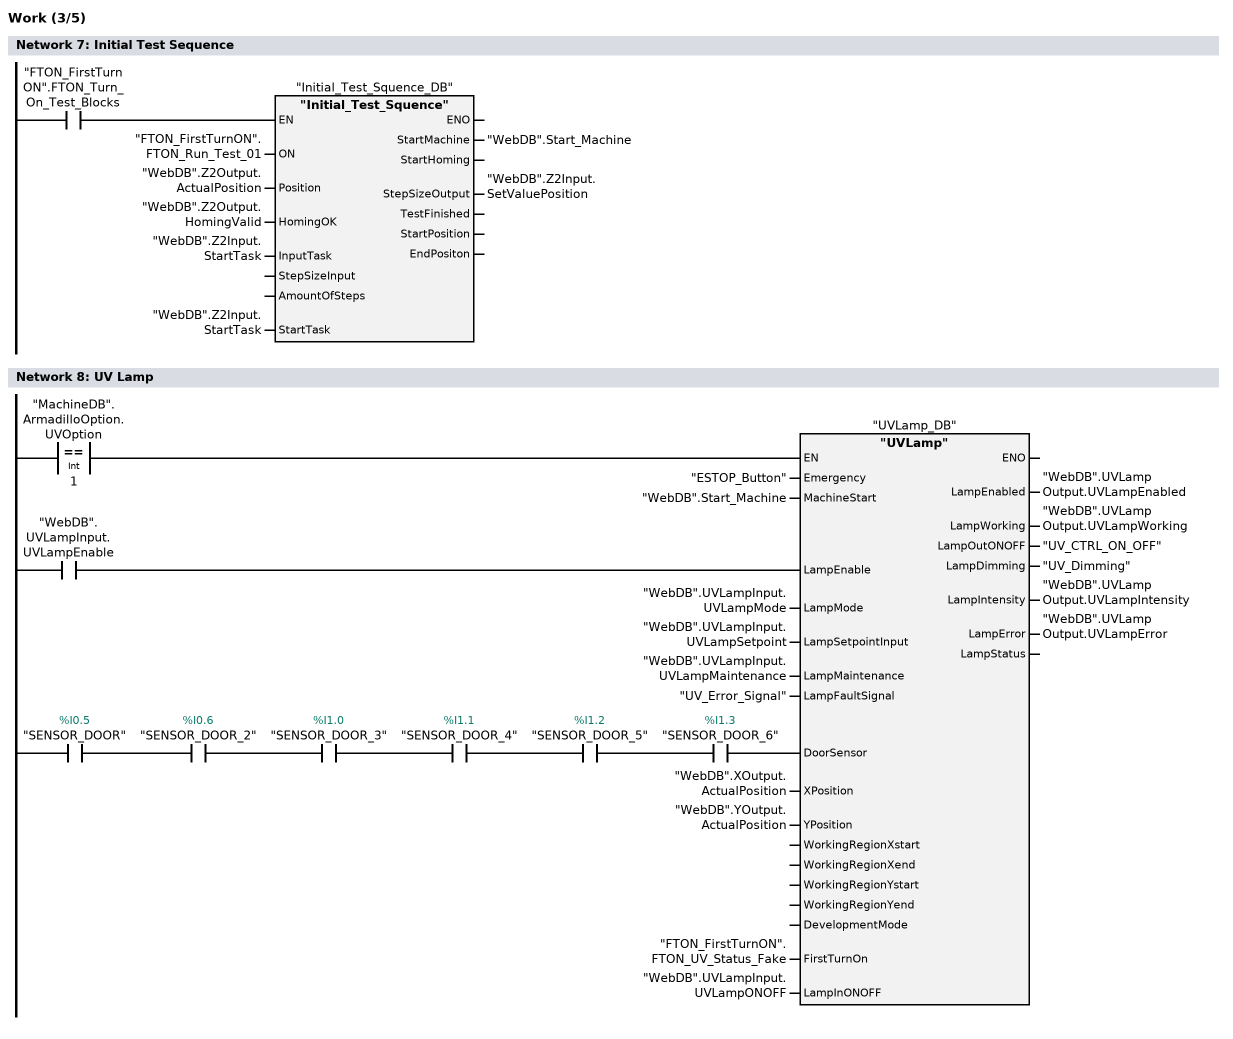
   RUNG wire#powerrail
      Contact( "FTON_FirstTurnON".FTON_Turn_On_Test_Blocks )
      "Initial_Test_Squence_DB"(ON := "FTON_FirstTurnON".FTON_Run_Test_01, Position := "WebDB".Z2Output.ActualPosition, HomingOK := "WebDB".Z2Output.HomingValid, InputTask := "WebDB".Z2Input.StartTask, StepSizeInput :=, AmountOfSteps :=, StartTask := "WebDB".Z2Input.StartTask, StartMachine => "WebDB".Start_Machine, StartHoming =>, StepSizeOutput => "WebDB".Z2Input.SetValuePosition, TestFinished =>, StartPosition =>, EndPositon =>)
   END_RUNG
   // the same network as SCL:
   IF "FTON_FirstTurnON".FTON_Turn_On_Test_Blocks THEN
       "Initial_Test_Squence_DB"(ON := "FTON_FirstTurnON".FTON_Run_Test_01,   // "Initial_Test_Squence"
                               Position := "WebDB".Z2Output.ActualPosition,
                               HomingOK := "WebDB".Z2Output.HomingValid,
                               InputTask := "WebDB".Z2Input.StartTask,
                               StartTask := "WebDB".Z2Input.StartTask,
                               StartMachine => "WebDB".Start_Machine,
                               StepSizeOutput => "WebDB".Z2Input.SetValuePosition);
   END_IF;
END_REGION

REGION Network 8: UV Lamp
   RUNG wire#powerrail
      { S7_Templates := "SrcType := Int" } EQ_Contact(in1 := "MachineDB".ArmadilloOption.UVOption, in2 := 1)
      "UVLamp_DB"(LampEnable := wire#w1, DoorSensor := wire#w2, Emergency := "ESTOP_Button", MachineStart := "WebDB".Start_Machine, LampMode := "WebDB".UVLampInput.UVLampMode, LampSetpointInput := "WebDB".UVLampInput.UVLampSetpoint, LampMaintenance := "WebDB".UVLampInput.UVLampMaintenance, LampFaultSignal := "UV_Error_Signal", XPosition := "WebDB".XOutput.ActualPosition, YPosition := "WebDB".YOutput.ActualPosition, WorkingRegionXstart :=, WorkingRegionXend :=, WorkingRegionYstart :=, WorkingRegionYend :=, DevelopmentMode :=, FirstTurnOn := "FTON_FirstTurnON".FTON_UV_Status_Fake, LampInONOFF := "WebDB".UVLampInput.UVLampONOFF, LampEnabled => "WebDB".UVLampOutput.UVLampEnabled, LampWorking => "WebDB".UVLampOutput.UVLampWorking, LampOutONOFF => "UV_CTRL_ON_OFF", LampDimming => "UV_Dimming", LampIntensity => "WebDB".UVLampOutput.UVLampIntensity, LampError => "WebDB".UVLampOutput.UVLampError, LampStatus =>)
   END_RUNG
   RUNG wire#powerrail
      Contact( "WebDB".UVLampInput.UVLampEnable )
   END_RUNG wire#w1
   RUNG wire#powerrail
      Contact( "SENSOR_DOOR" )
      Contact( "SENSOR_DOOR_2" )
      Contact( "SENSOR_DOOR_3" )
      Contact( "SENSOR_DOOR_4" )
      Contact( "SENSOR_DOOR_5" )
      Contact( "SENSOR_DOOR_6" )
   END_RUNG wire#w2
   // the same network as SCL:
   IF "MachineDB".ArmadilloOption.UVOption = 1 THEN
       "UVLamp_DB"(Emergency := "ESTOP_Button",   // "UVLamp"
                   MachineStart := "WebDB".Start_Machine,
                   LampEnable := "WebDB".UVLampInput.UVLampEnable,
                   LampMode := "WebDB".UVLampInput.UVLampMode,
                   LampSetpointInput := "WebDB".UVLampInput.UVLampSetpoint,
                   LampMaintenance := "WebDB".UVLampInput.UVLampMaintenance,
                   LampFaultSignal := "UV_Error_Signal",
                   DoorSensor := "SENSOR_DOOR" AND "SENSOR_DOOR_2" AND "SENSOR_DOOR_3" AND "SENSOR_DOOR_4" AND "SENSOR_DOOR_5" AND "SENSOR_DOOR_6",
                   XPosition := "WebDB".XOutput.ActualPosition,
                   YPosition := "WebDB".YOutput.ActualPosition,
                   FirstTurnOn := "FTON_FirstTurnON".FTON_UV_Status_Fake,
                   LampInONOFF := "WebDB".UVLampInput.UVLampONOFF,
                   LampEnabled => "WebDB".UVLampOutput.UVLampEnabled,
                   LampWorking => "WebDB".UVLampOutput.UVLampWorking,
                   LampOutONOFF => "UV_CTRL_ON_OFF",
                   LampDimming => "UV_Dimming",
                   LampIntensity => "WebDB".UVLampOutput.UVLampIntensity,
                   LampError => "WebDB".UVLampOutput.UVLampError);
   END_IF;
END_REGION

REGION Network 9: Stacklight
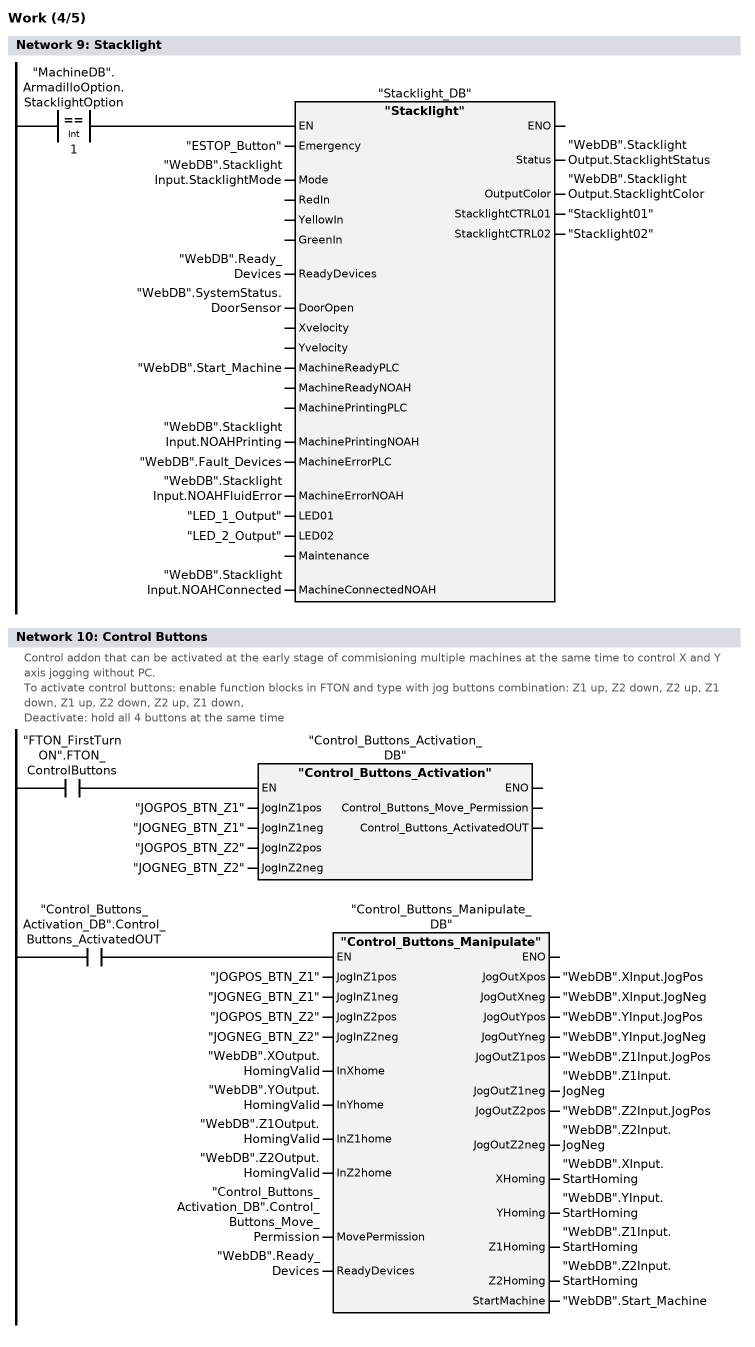
   RUNG wire#powerrail
      { S7_Templates := "SrcType := Int" } EQ_Contact(in1 := "MachineDB".ArmadilloOption.StacklightOption, in2 := 1)
      "Stacklight_DB"(Emergency := "ESTOP_Button", Mode := "WebDB".StacklightInput.StacklightMode, RedIn :=, YellowIn :=, GreenIn :=, ReadyDevices := "WebDB".Ready_Devices, DoorOpen := "WebDB".SystemStatus.DoorSensor, Xvelocity :=, Yvelocity :=, MachineReadyPLC := "WebDB".Start_Machine, MachineReadyNOAH :=, MachinePrintingPLC :=, MachinePrintingNOAH := "WebDB".StacklightInput.NOAHPrinting, MachineErrorPLC := "WebDB".Fault_Devices, MachineErrorNOAH := "WebDB".StacklightInput.NOAHFluidError, LED01 := "LED_1_Output", LED02 := "LED_2_Output", Maintenance :=, MachineConnectedNOAH := "WebDB".StacklightInput.NOAHConnected, Status => "WebDB".StacklightOutput.StacklightStatus, OutputColor => "WebDB".StacklightOutput.StacklightColor, StacklightCTRL01 => "Stacklight01", StacklightCTRL02 => "Stacklight02")
   END_RUNG
   // the same network as SCL:
   IF "MachineDB".ArmadilloOption.StacklightOption = 1 THEN
       "Stacklight_DB"(Emergency := "ESTOP_Button",   // "Stacklight"
                       Mode := "WebDB".StacklightInput.StacklightMode,
                       ReadyDevices := "WebDB".Ready_Devices,
                       DoorOpen := "WebDB".SystemStatus.DoorSensor,
                       MachineReadyPLC := "WebDB".Start_Machine,
                       MachinePrintingNOAH := "WebDB".StacklightInput.NOAHPrinting,
                       MachineErrorPLC := "WebDB".Fault_Devices,
                       MachineErrorNOAH := "WebDB".StacklightInput.NOAHFluidError,
                       LED01 := "LED_1_Output",
                       LED02 := "LED_2_Output",
                       MachineConnectedNOAH := "WebDB".StacklightInput.NOAHConnected,
                       Status => "WebDB".StacklightOutput.StacklightStatus,
                       OutputColor => "WebDB".StacklightOutput.StacklightColor,
                       StacklightCTRL01 => "Stacklight01",
                       StacklightCTRL02 => "Stacklight02");
   END_IF;
END_REGION

REGION Network 10: Control Buttons
   // Control addon that can be activated at the early stage of commisioning multiple machines at the same time to control X and Y axis jogging without PC.
   // 
   // To activate control buttons: enable function blocks in FTON and type with jog buttons combination: Z1 up, Z2 down, Z2 up, Z1 down, Z1 up, Z2 down, Z2 up, Z1 down,
   // 
   // Deactivate: hold all 4 buttons at the same time
   RUNG wire#powerrail
      Contact( "FTON_FirstTurnON".FTON_ControlButtons )
      "Control_Buttons_Activation_DB"(JogInZ1pos := "JOGPOS_BTN_Z1", JogInZ1neg := "JOGNEG_BTN_Z1", JogInZ2pos := "JOGPOS_BTN_Z2", JogInZ2neg := "JOGNEG_BTN_Z2", Control_Buttons_Move_Permission =>, Control_Buttons_ActivatedOUT =>)
   END_RUNG
   RUNG wire#powerrail
      Contact( "Control_Buttons_Activation_DB".Control_Buttons_ActivatedOUT )
      "Control_Buttons_Manipulate_DB"(JogInZ1pos := "JOGPOS_BTN_Z1", JogInZ1neg := "JOGNEG_BTN_Z1", JogInZ2pos := "JOGPOS_BTN_Z2", JogInZ2neg := "JOGNEG_BTN_Z2", InXhome := "WebDB".XOutput.HomingValid, InYhome := "WebDB".YOutput.HomingValid, InZ1home := "WebDB".Z1Output.HomingValid, InZ2home := "WebDB".Z2Output.HomingValid, MovePermission := "Control_Buttons_Activation_DB".Control_Buttons_Move_Permission, ReadyDevices := "WebDB".Ready_Devices, JogOutXpos => "WebDB".XInput.JogPos, JogOutXneg => "WebDB".XInput.JogNeg, JogOutYpos => "WebDB".YInput.JogPos, JogOutYneg => "WebDB".YInput.JogNeg, JogOutZ1pos => "WebDB".Z1Input.JogPos, JogOutZ1neg => "WebDB".Z1Input.JogNeg, JogOutZ2pos => "WebDB".Z2Input.JogPos, JogOutZ2neg => "WebDB".Z2Input.JogNeg, XHoming => "WebDB".XInput.StartHoming, YHoming => "WebDB".YInput.StartHoming, Z1Homing => "WebDB".Z1Input.StartHoming, Z2Homing => "WebDB".Z2Input.StartHoming, StartMachine => "WebDB".Start_Machine)
   END_RUNG
   // the same network as SCL:
   IF "FTON_FirstTurnON".FTON_ControlButtons THEN
       "Control_Buttons_Activation_DB"(JogInZ1pos := "JOGPOS_BTN_Z1",   // "Control_Buttons_Activation"
                               JogInZ1neg := "JOGNEG_BTN_Z1",
                               JogInZ2pos := "JOGPOS_BTN_Z2",
                               JogInZ2neg := "JOGNEG_BTN_Z2");
   END_IF;
   IF "Control_Buttons_Activation_DB".Control_Buttons_ActivatedOUT THEN
       "Control_Buttons_Manipulate_DB"(JogInZ1pos := "JOGPOS_BTN_Z1",   // "Control_Buttons_Manipulate"
                               JogInZ1neg := "JOGNEG_BTN_Z1",
                               JogInZ2pos := "JOGPOS_BTN_Z2",
                               JogInZ2neg := "JOGNEG_BTN_Z2",
                               InXhome := "WebDB".XOutput.HomingValid,
                               InYhome := "WebDB".YOutput.HomingValid,
                               InZ1home := "WebDB".Z1Output.HomingValid,
                               InZ2home := "WebDB".Z2Output.HomingValid,
                               MovePermission := "Control_Buttons_Activation_DB".Control_Buttons_Move_Permission,
                               ReadyDevices := "WebDB".Ready_Devices,
                               JogOutXpos => "WebDB".XInput.JogPos,
                               JogOutXneg => "WebDB".XInput.JogNeg,
                               JogOutYpos => "WebDB".YInput.JogPos,
                               JogOutYneg => "WebDB".YInput.JogNeg,
                               JogOutZ1pos => "WebDB".Z1Input.JogPos,
                               JogOutZ1neg => "WebDB".Z1Input.JogNeg,
                               JogOutZ2pos => "WebDB".Z2Input.JogPos,
                               JogOutZ2neg => "WebDB".Z2Input.JogNeg,
                               XHoming => "WebDB".XInput.StartHoming,
                               YHoming => "WebDB".YInput.StartHoming,
                               Z1Homing => "WebDB".Z1Input.StartHoming,
                               Z2Homing => "WebDB".Z2Input.StartHoming,
                               StartMachine => "WebDB".Start_Machine);
   END_IF;
END_REGION

REGION Network 11: Data Logging
   // Details to start the logging process:
   // 1) Activate web server
   // 2) Set variables to log by assigning them to DataLogging block inputs
   // 3) Create logging file in the FTON
   // 4) Start logging in the FTON
   // 5) Download the file via web server
   // 
   // There is a limited amount of data that can be written due to limited memory capacity. The file will be overwritten after certain amount of records. It is possible to create a new file based on amount of records, should be developed in the future.
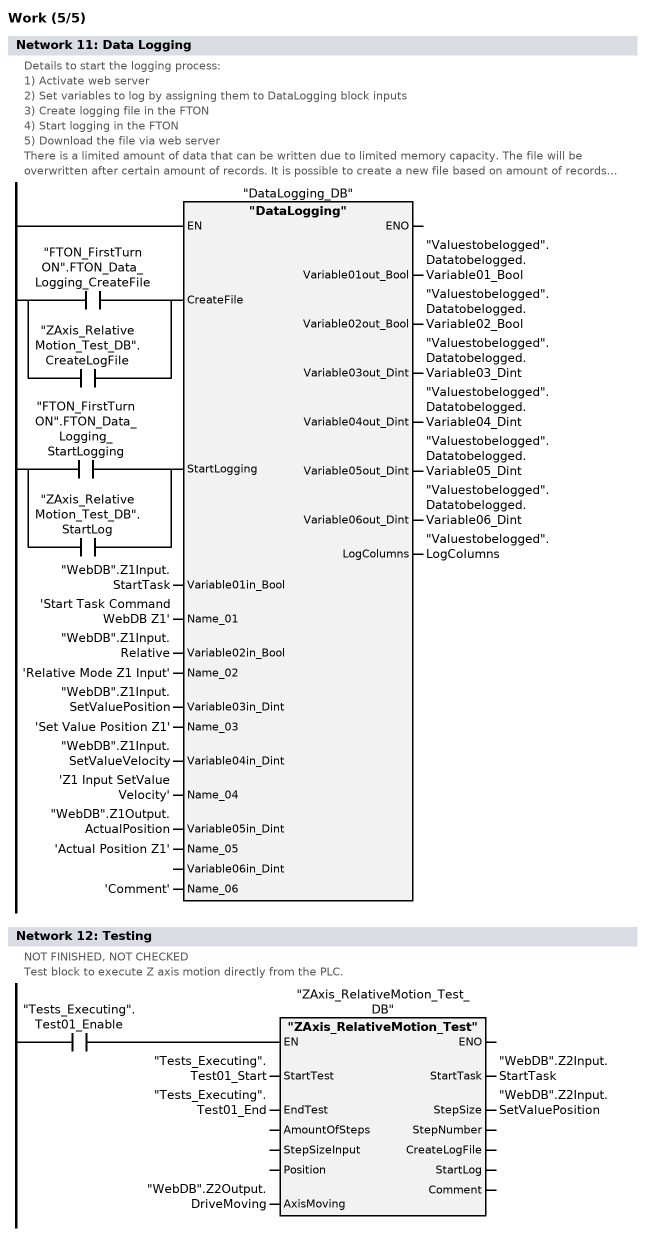
   RUNG wire#powerrail
      "DataLogging_DB"(CreateFile := wire#w1, StartLogging := wire#w2, Variable01in_Bool := "WebDB".Z1Input.StartTask, Name_01 := 'Start Task Command WebDB Z1', Variable02in_Bool := "WebDB".Z1Input.Relative, Name_02 := 'Relative Mode Z1 Input', Variable03in_Dint := "WebDB".Z1Input.SetValuePosition, Name_03 := 'Set Value Position Z1', Variable04in_Dint := "WebDB".Z1Input.SetValueVelocity, Name_04 := 'Z1 Input SetValueVelocity', Variable05in_Dint := "WebDB".Z1Output.ActualPosition, Name_05 := 'Actual Position Z1', Variable06in_Dint :=, Name_06 := 'Comment', Variable01out_Bool => "Valuestobelogged".Datatobelogged.Variable01_Bool, Variable02out_Bool => "Valuestobelogged".Datatobelogged.Variable02_Bool, Variable03out_Dint => "Valuestobelogged".Datatobelogged.Variable03_Dint, Variable04out_Dint => "Valuestobelogged".Datatobelogged.Variable04_Dint, Variable05out_Dint => "Valuestobelogged".Datatobelogged.Variable05_Dint, Variable06out_Dint => "Valuestobelogged".Datatobelogged.Variable06_Dint, LogColumns => "Valuestobelogged".LogColumns)
   END_RUNG
   RUNG wire#powerrail
      Contact( "FTON_FirstTurnON".FTON_Data_Logging_CreateFile )
   END_RUNG wire#w1
   RUNG wire#powerrail
      Contact( "ZAxis_RelativeMotion_Test_DB".CreateLogFile )
   END_RUNG wire#w1
   RUNG wire#powerrail
      Contact( "FTON_FirstTurnON".FTON_Data_Logging_StartLogging )
   END_RUNG wire#w2
   RUNG wire#powerrail
      Contact( "ZAxis_RelativeMotion_Test_DB".StartLog )
   END_RUNG wire#w2
   // the same network as SCL:
   "DataLogging_DB"(CreateFile := "FTON_FirstTurnON".FTON_Data_Logging_CreateFile OR "ZAxis_RelativeMotion_Test_DB".CreateLogFile,   // "DataLogging"
                    StartLogging := "FTON_FirstTurnON".FTON_Data_Logging_StartLogging OR "ZAxis_RelativeMotion_Test_DB".StartLog,
                    Variable01in_Bool := "WebDB".Z1Input.StartTask,
                    Name_01 := 'Start Task Command WebDB Z1',
                    Variable02in_Bool := "WebDB".Z1Input.Relative,
                    Name_02 := 'Relative Mode Z1 Input',
                    Variable03in_Dint := "WebDB".Z1Input.SetValuePosition,
                    Name_03 := 'Set Value Position Z1',
                    Variable04in_Dint := "WebDB".Z1Input.SetValueVelocity,
                    Name_04 := 'Z1 Input SetValueVelocity',
                    Variable05in_Dint := "WebDB".Z1Output.ActualPosition,
                    Name_05 := 'Actual Position Z1',
                    Name_06 := 'Comment',
                    Variable01out_Bool => "Valuestobelogged".Datatobelogged.Variable01_Bool,
                    Variable02out_Bool => "Valuestobelogged".Datatobelogged.Variable02_Bool,
                    Variable03out_Dint => "Valuestobelogged".Datatobelogged.Variable03_Dint,
                    Variable04out_Dint => "Valuestobelogged".Datatobelogged.Variable04_Dint,
                    Variable05out_Dint => "Valuestobelogged".Datatobelogged.Variable05_Dint,
                    Variable06out_Dint => "Valuestobelogged".Datatobelogged.Variable06_Dint,
                    LogColumns => "Valuestobelogged".LogColumns);
END_REGION

REGION Network 12: Testing
   // NOT FINISHED, NOT CHECKED
   // Test block to execute Z axis motion directly from the PLC.
   RUNG wire#powerrail
      Contact( "Tests_Executing".Test01_Enable )
      "ZAxis_RelativeMotion_Test_DB"(StartTest := "Tests_Executing".Test01_Start, EndTest := "Tests_Executing".Test01_End, AmountOfSteps :=, StepSizeInput :=, Position :=, AxisMoving := "WebDB".Z2Output.DriveMoving, StartTask => "WebDB".Z2Input.StartTask, StepSize => "WebDB".Z2Input.SetValuePosition, StepNumber =>, CreateLogFile =>, StartLog =>, Comment =>)
   END_RUNG
   // the same network as SCL:
   IF "Tests_Executing".Test01_Enable THEN
       "ZAxis_RelativeMotion_Test_DB"(StartTest := "Tests_Executing".Test01_Start,   // "ZAxis_RelativeMotion_Test"
                               EndTest := "Tests_Executing".Test01_End,
                               AxisMoving := "WebDB".Z2Output.DriveMoving,
                               StartTask => "WebDB".Z2Input.StartTask,
                               StepSize => "WebDB".Z2Input.SetValuePosition);
   END_IF;
END_REGION
END_ORGANIZATION_BLOCK

FUNCTION "Enable_machine" : Void   // FC5, LAD
{ S7_Optimized_Access := 'TRUE' }
VERSION : 0.1
BEGIN

REGION Network 1: Halt Axis
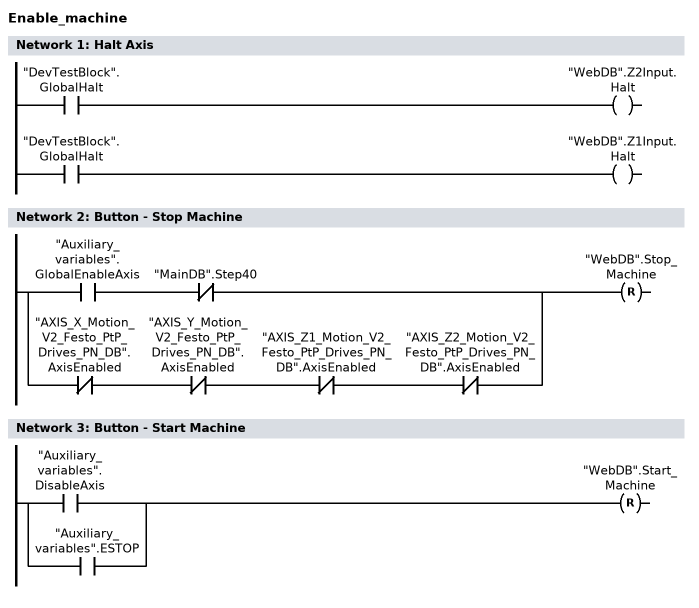
   RUNG wire#powerrail
      Contact( "DevTestBlock".GlobalHalt )
      Coil( "WebDB".Z2Input.Halt )
   END_RUNG
   RUNG wire#powerrail
      Contact( "DevTestBlock".GlobalHalt )
      Coil( "WebDB".Z1Input.Halt )
   END_RUNG
   // the same network as SCL:
   "WebDB".Z2Input.Halt := "DevTestBlock".GlobalHalt;
   "WebDB".Z1Input.Halt := "DevTestBlock".GlobalHalt;
END_REGION

REGION Network 2: Button - Stop Machine
   RUNG wire#powerrail
      Contact( "Auxiliary_variables".GlobalEnableAxis )
      I_Contact( "MainDB".Step40 )
      wire#w1
      R_Coil( "WebDB".Stop_Machine )
   END_RUNG
   RUNG wire#powerrail
      I_Contact( "AXIS_X_Motion_V2_Festo_PtP_Drives_PN_DB".AxisEnabled )
      I_Contact( "AXIS_Y_Motion_V2_Festo_PtP_Drives_PN_DB".AxisEnabled )
      I_Contact( "AXIS_Z1_Motion_V2_Festo_PtP_Drives_PN_DB".AxisEnabled )
      I_Contact( "AXIS_Z2_Motion_V2_Festo_PtP_Drives_PN_DB".AxisEnabled )
   END_RUNG wire#w1
   // the same network as SCL:
   IF ("Auxiliary_variables".GlobalEnableAxis AND NOT "MainDB".Step40) OR (NOT "AXIS_X_Motion_V2_Festo_PtP_Drives_PN_DB".AxisEnabled AND NOT "AXIS_Y_Motion_V2_Festo_PtP_Drives_PN_DB".AxisEnabled AND NOT "AXIS_Z1_Motion_V2_Festo_PtP_Drives_PN_DB".AxisEnabled AND NOT "AXIS_Z2_Motion_V2_Festo_PtP_Drives_PN_DB".AxisEnabled) THEN
       "WebDB".Stop_Machine := FALSE;
   END_IF;
END_REGION

REGION Network 3: Button - Start Machine
   RUNG wire#powerrail
      Contact( "Auxiliary_variables".DisableAxis )
      wire#w1
      R_Coil( "WebDB".Start_Machine )
   END_RUNG
   RUNG wire#powerrail
      Contact( "Auxiliary_variables".ESTOP )
   END_RUNG wire#w1
   // the same network as SCL:
   IF "Auxiliary_variables".DisableAxis OR "Auxiliary_variables".ESTOP THEN
       "WebDB".Start_Machine := FALSE;
   END_IF;
END_REGION
END_FUNCTION

FUNCTION_BLOCK "IR_Heater_Control"   // FB17, LAD
TITLE = Description
{ S7_Optimized_Access := 'TRUE' }
VERSION : 0.1
// How to control and set the IR lamp:
// To turn on the IR lamp the machine needs to be started and the doors closed. Heater setpoint should be set from 0-100 "Heater_Setpoint", lamp should be turned on by "Heater_ON_OFF". The lamp will activate only when the certain conditions are meet (position/direction/time).
// 
// Right now, the signal from NOAH is being send when spreading and the permission for the lamp is being keep in the function block for a certain period of time to enable the lamp on the way back.
// 
// E-STOP - always check!
// 
// Modes:
// 0 - Heating Feedbox/Printbox when spreading and executing the heater on the way back from PLC
// 1 - Heating only on the way back from NOAH
// 
// Safety is based only on timer. Hardware protection should be implemented ASAP (contactor controlled by thermal fuse / thermistor to cut off the power if the temperature exceeds certain level).
// 
// Things to implement:
// - Remote temperature sensor(already purchased some time ago).
// - Heater_MathFunction to operate heater better based on the measured results
// - PID control
// 
// Status:
// Filip 14.12.2022: Added modes to give full control to NOAH (Mode 1) or control heater on the way back from PLC (Mode 0)
   VAR_INPUT
      MachineNumber : Int;
      Mode : Int := 1;   // 0 - Heating partly from PLC; 1 - Full control from NOAH
      DoorSenor : Bool;
      RollerON : Bool;   // General heater safety condition
      Heater_Safety_PDL : Real;   // Pulse Duration Limit - set by technician or engineer in charge, don't change
      Heater_PWM_address : HW_PWM;   // PLC PWM output address
      Heater_Setpoint : Real;
      "E-STOP" : Bool;
      Heater_ON_OFF : Bool;   // WebDB
      FeedboxHeating : Bool;
      PrintboxHeating : Bool;
      AxisYActualPosition : DInt;
      AxisYActualVelocity : Real;
      FeedboxStartMachine : DInt;
      FeedboxEndMachine : DInt;
      PrintboxStartMachine : DInt;
      PrintboxEndMachine : DInt;
      HeaterTest : Bool;
   END_VAR
   VAR_OUTPUT
      Heater_Output : Bool;
      Heater_Pulse_Duration : Int;
      Heater_Error : Int;
      Heater_Output_Check : Int;
      RollerONWayBack : Bool;
      WrongPositionInput : Bool;
   END_VAR
   VAR
      Heater_Scale_LimitReductionBed : Real := 1000.0;   // For big printbox set 70.0, for testing and reduction bed set 100.0
      Heater_Scale_LimitNoReduction : Real := 700.0;
      Heater_Scale_Internal : Real;
      Heater_status : Bool := false;
      Heater_signal : Int;
      Heater_safety_input : Bool := true;   // General heater safety condition
      Heater_error_code : Word;   // Error codes: 0 - OK; 80A1 - Hardware ID; 80D0 - PWM not activated
      Heater_Output_Check_1 : Int;
      SafetyTime : Bool;   // Safety time to not overheat recoater
      ReverseDirectionPermission : Bool := false;   // Permission for using IR on the way back
      ReverseDirection : Bool;
      HeaterStatusSave : Bool;
      HeaterStatusTimeExpired : Bool;
      TurningOnInAdvanceSTART : DInt := 150000;
      TurningOnInAdvanceEND : DInt := 225000;
      TurningOnInAdvanceRefresh : DInt := 2000;
      Position : DInt;
      FeedboxHeatingON : Bool := false;
      PrintboxHeatingON : Bool := true;
      HeaterWayBack : Bool := true;
      MaintenanceSkipPositionPermission : Bool;
      MaintenanceSkipRoller : Bool;
      DevModeHeater : Bool;
      DevelopmentAddOn01 : Bool;   // For testing - Will be removed when checked
   END_VAR
   VAR_TEMP
      Heater_SetpointTemp : Int;
      Heater_SetpointOneThird : Int;
      InitialOneThird : Bool;
      Heater_PDLTemp : Int;
      Heater_PDL_conv : Real;
      Heater_Setpoint_Internal01 : Real;
      Heater_Setpoint_Internal02 : Real;
      Heater_Overload : Bool;
      PositionPermissionRight : Bool;
      PositionPermissionLeft : Bool;
      VelocityFactor : Real;
      PositionStartInternal : DInt;
      PositionStartInAdvance : DInt;
      PositionEndInternal : DInt;
      PositionEndInAdvance : DInt;
      PositionEndRefresh : DInt;
      PrintboxSize : DInt;
   END_VAR
   VAR_TEMP   // added for the SCL form of the ladder/FBD networks
      _w1 : Bool;
   END_VAR
BEGIN

REGION Network 1: Safety
   // Heater time safety limitation to avoid overheating parts.
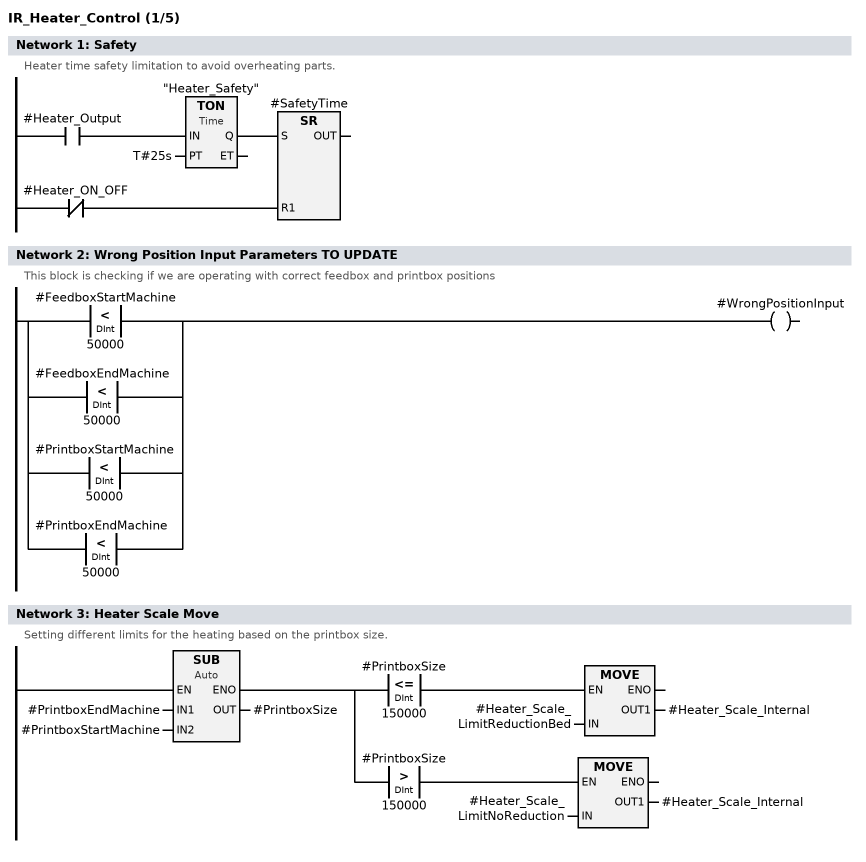
   RUNG wire#powerrail
      Contact( #Heater_Output )
      { S7_Templates := "time_type := Time" } "Heater_Safety".TON(pt := T#25s, et =>)
      S_SR(operand := #SafetyTime, r1 := wire#w1)
   END_RUNG
   RUNG wire#powerrail
      I_Contact( #Heater_ON_OFF )
   END_RUNG wire#w1
   // the same network as SCL:
   "Heater_Safety".TON(IN := #Heater_Output, PT := T#25s);
   IF "Heater_Safety".Q THEN
       #SafetyTime := TRUE;   // SR flip-flop
   END_IF;
   IF NOT #Heater_ON_OFF THEN #SafetyTime := FALSE; END_IF;
END_REGION

REGION Network 2: Wrong Position Input Parameters TO UPDATE
   // This block is checking if we are operating with correct feedbox and printbox positions
   RUNG wire#powerrail
      { S7_Templates := "SrcType := DInt" } LT_Contact(in1 := #FeedboxStartMachine, in2 := 50000)
      wire#w1
      Coil( #WrongPositionInput )
   END_RUNG
   RUNG wire#powerrail
      { S7_Templates := "SrcType := DInt" } LT_Contact(in1 := #FeedboxEndMachine, in2 := 50000)
   END_RUNG wire#w1
   RUNG wire#powerrail
      { S7_Templates := "SrcType := DInt" } LT_Contact(in1 := #PrintboxStartMachine, in2 := 50000)
   END_RUNG wire#w1
   RUNG wire#powerrail
      { S7_Templates := "SrcType := DInt" } LT_Contact(in1 := #PrintboxEndMachine, in2 := 50000)
   END_RUNG wire#w1
   // the same network as SCL:
   #WrongPositionInput := (#FeedboxStartMachine < 50000) OR (#FeedboxEndMachine < 50000) OR (#PrintboxStartMachine < 50000) OR (#PrintboxEndMachine < 50000);
END_REGION

REGION Network 3: Heater Scale Move
   // Setting different limits for the heating based on the printbox size.
   RUNG wire#powerrail
      Sub(in1 := #PrintboxEndMachine, in2 := #PrintboxStartMachine, out => #PrintboxSize)
      wire#w1
      { S7_Templates := "SrcType := DInt" } LE_Contact(in1 := #PrintboxSize, in2 := 150000)
      Move(in := #Heater_Scale_LimitReductionBed, out1 => #Heater_Scale_Internal)
   END_RUNG
   RUNG wire#w1
      { S7_Templates := "SrcType := DInt" } GT_Contact(in1 := #PrintboxSize, in2 := 150000)
      Move(in := #Heater_Scale_LimitNoReduction, out1 => #Heater_Scale_Internal)
   END_RUNG
   // the same network as SCL:
   #PrintboxSize := #PrintboxEndMachine - #PrintboxStartMachine;
   IF #PrintboxSize <= 150000 THEN #Heater_Scale_Internal := #Heater_Scale_LimitReductionBed; END_IF;
   IF #PrintboxSize > 150000 THEN #Heater_Scale_Internal := #Heater_Scale_LimitNoReduction; END_IF;
END_REGION

REGION Network 4: Positions In Advance
   // Calculation of positions to turn on IR lamp in advance, due to long rise time.
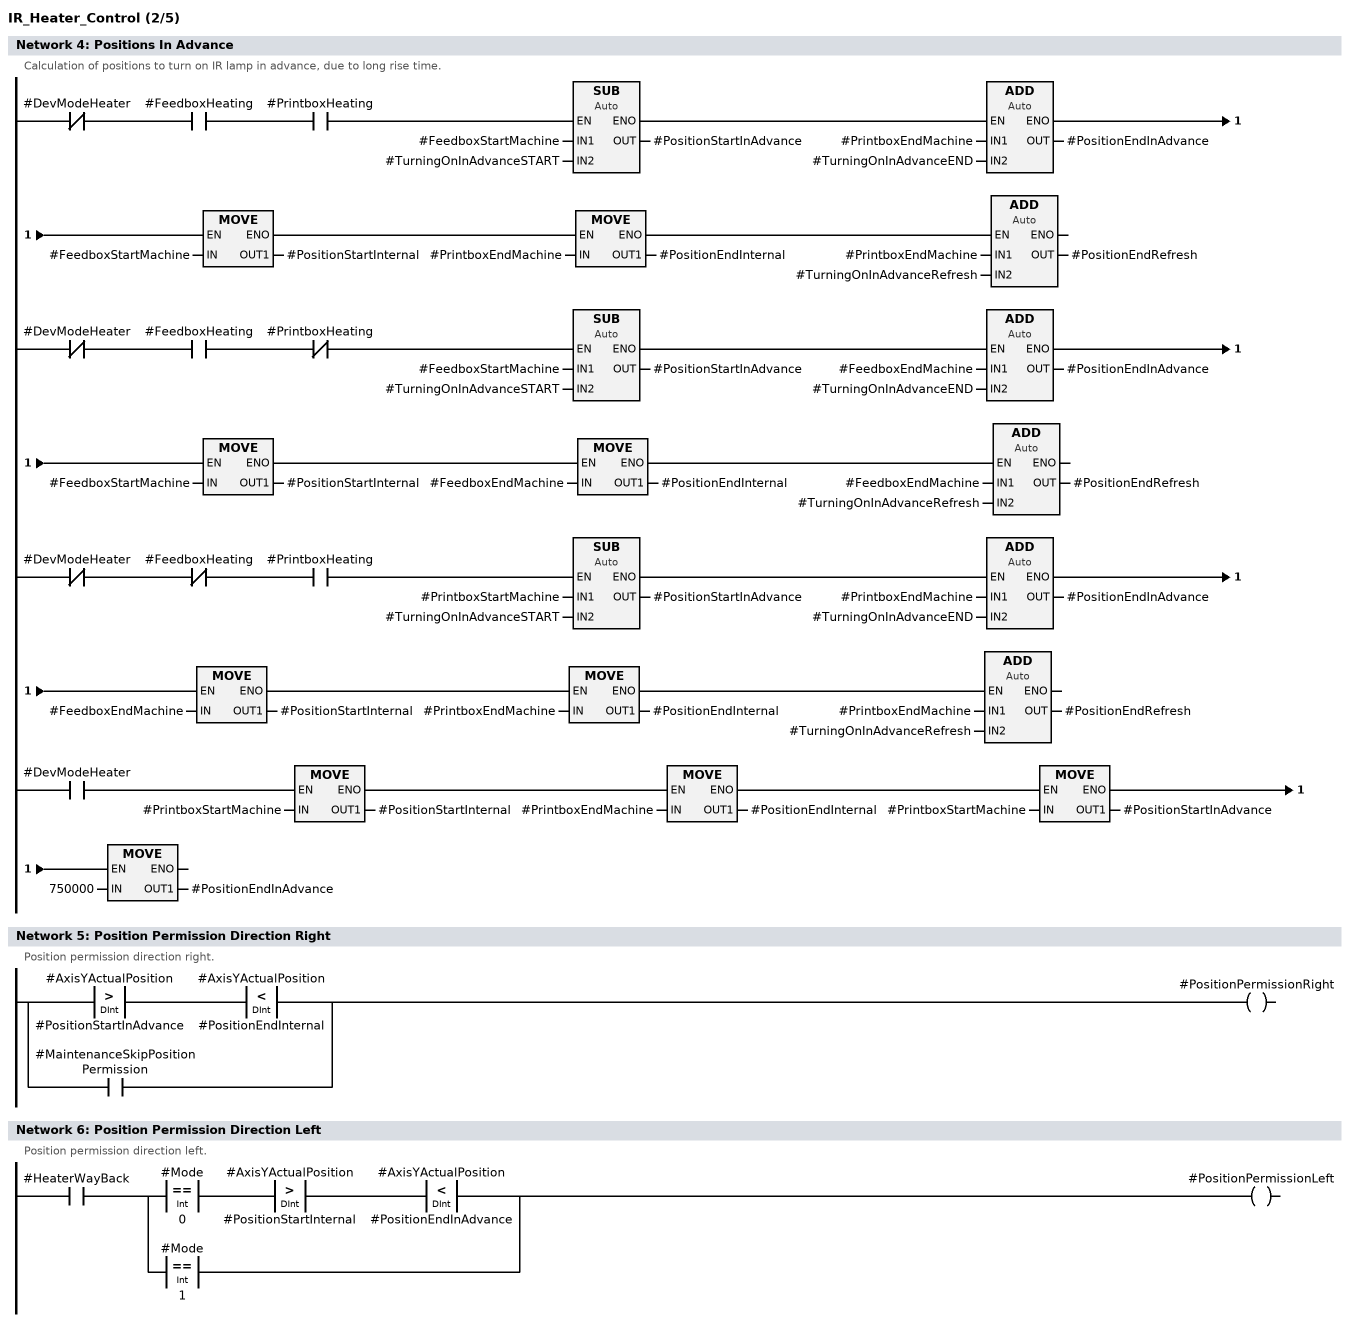
   RUNG wire#powerrail
      I_Contact( #DevModeHeater )
      Contact( #FeedboxHeating )
      Contact( #PrintboxHeating )
      Sub(in1 := #FeedboxStartMachine, in2 := #TurningOnInAdvanceSTART, out => #PositionStartInAdvance)
      Add(in1 := #PrintboxEndMachine, in2 := #TurningOnInAdvanceEND, out => #PositionEndInAdvance)
      Move(in := #FeedboxStartMachine, out1 => #PositionStartInternal)
      Move(in := #PrintboxEndMachine, out1 => #PositionEndInternal)
      Add(in1 := #PrintboxEndMachine, in2 := #TurningOnInAdvanceRefresh, out => #PositionEndRefresh)
   END_RUNG
   RUNG wire#powerrail
      I_Contact( #DevModeHeater )
      Contact( #FeedboxHeating )
      I_Contact( #PrintboxHeating )
      Sub(in1 := #FeedboxStartMachine, in2 := #TurningOnInAdvanceSTART, out => #PositionStartInAdvance)
      Add(in1 := #FeedboxEndMachine, in2 := #TurningOnInAdvanceEND, out => #PositionEndInAdvance)
      Move(in := #FeedboxStartMachine, out1 => #PositionStartInternal)
      Move(in := #FeedboxEndMachine, out1 => #PositionEndInternal)
      Add(in1 := #FeedboxEndMachine, in2 := #TurningOnInAdvanceRefresh, out => #PositionEndRefresh)
   END_RUNG
   RUNG wire#powerrail
      I_Contact( #DevModeHeater )
      I_Contact( #FeedboxHeating )
      Contact( #PrintboxHeating )
      Sub(in1 := #PrintboxStartMachine, in2 := #TurningOnInAdvanceSTART, out => #PositionStartInAdvance)
      Add(in1 := #PrintboxEndMachine, in2 := #TurningOnInAdvanceEND, out => #PositionEndInAdvance)
      Move(in := #FeedboxEndMachine, out1 => #PositionStartInternal)
      Move(in := #PrintboxEndMachine, out1 => #PositionEndInternal)
      Add(in1 := #PrintboxEndMachine, in2 := #TurningOnInAdvanceRefresh, out => #PositionEndRefresh)
   END_RUNG
   RUNG wire#powerrail
      Contact( #DevModeHeater )
      Move(in := #PrintboxStartMachine, out1 => #PositionStartInternal)
      Move(in := #PrintboxEndMachine, out1 => #PositionEndInternal)
      Move(in := #PrintboxStartMachine, out1 => #PositionStartInAdvance)
      Move(in := 750000, out1 => #PositionEndInAdvance)
   END_RUNG
   // the same network as SCL:
   IF NOT #DevModeHeater AND #FeedboxHeating AND #PrintboxHeating THEN
       #PositionStartInAdvance := #FeedboxStartMachine - #TurningOnInAdvanceSTART;
       #PositionEndInAdvance := #PrintboxEndMachine + #TurningOnInAdvanceEND;
       #PositionStartInternal := #FeedboxStartMachine;
       #PositionEndInternal := #PrintboxEndMachine;
       #PositionEndRefresh := #PrintboxEndMachine + #TurningOnInAdvanceRefresh;
   END_IF;
   IF NOT #DevModeHeater AND #FeedboxHeating AND NOT #PrintboxHeating THEN
       #PositionStartInAdvance := #FeedboxStartMachine - #TurningOnInAdvanceSTART;
       #PositionEndInAdvance := #FeedboxEndMachine + #TurningOnInAdvanceEND;
       #PositionStartInternal := #FeedboxStartMachine;
       #PositionEndInternal := #FeedboxEndMachine;
       #PositionEndRefresh := #FeedboxEndMachine + #TurningOnInAdvanceRefresh;
   END_IF;
   IF NOT #DevModeHeater AND NOT #FeedboxHeating AND #PrintboxHeating THEN
       #PositionStartInAdvance := #PrintboxStartMachine - #TurningOnInAdvanceSTART;
       #PositionEndInAdvance := #PrintboxEndMachine + #TurningOnInAdvanceEND;
       #PositionStartInternal := #FeedboxEndMachine;
       #PositionEndInternal := #PrintboxEndMachine;
       #PositionEndRefresh := #PrintboxEndMachine + #TurningOnInAdvanceRefresh;
   END_IF;
   IF #DevModeHeater THEN
       #PositionStartInternal := #PrintboxStartMachine;
       #PositionEndInternal := #PrintboxEndMachine;
       #PositionStartInAdvance := #PrintboxStartMachine;
       #PositionEndInAdvance := 750000;
   END_IF;
END_REGION

REGION Network 5: Position Permission Direction Right
   // Position permission direction right.
   RUNG wire#powerrail
      { S7_Templates := "SrcType := DInt" } GT_Contact(in1 := #AxisYActualPosition, in2 := #PositionStartInAdvance)
      { S7_Templates := "SrcType := DInt" } LT_Contact(in1 := #AxisYActualPosition, in2 := #PositionEndInternal)
      wire#w1
      Coil( #PositionPermissionRight )
   END_RUNG
   RUNG wire#powerrail
      Contact( #MaintenanceSkipPositionPermission )
   END_RUNG wire#w1
   // the same network as SCL:
   #PositionPermissionRight := ((#AxisYActualPosition > #PositionStartInAdvance) AND (#AxisYActualPosition < #PositionEndInternal)) OR #MaintenanceSkipPositionPermission;
END_REGION

REGION Network 6: Position Permission Direction Left
   // Position permission direction left.
   RUNG wire#powerrail
      Contact( #HeaterWayBack )
      wire#w1
      { S7_Templates := "SrcType := Int" } EQ_Contact(in1 := #Mode, in2 := 0)
      { S7_Templates := "SrcType := DInt" } GT_Contact(in1 := #AxisYActualPosition, in2 := #PositionStartInternal)
      { S7_Templates := "SrcType := DInt" } LT_Contact(in1 := #AxisYActualPosition, in2 := #PositionEndInAdvance)
      wire#w2
      Coil( #PositionPermissionLeft )
   END_RUNG
   RUNG wire#w1
      { S7_Templates := "SrcType := Int" } EQ_Contact(in1 := #Mode, in2 := 1)
   END_RUNG wire#w2
   // the same network as SCL:
   #PositionPermissionLeft := #HeaterWayBack AND (((#Mode = 0) AND (#AxisYActualPosition > #PositionStartInternal) AND (#AxisYActualPosition < #PositionEndInAdvance)) OR (#Mode = 1));
END_REGION

REGION Network 7: Reverse Direction for Armadillo V6
   // Detection of the reverse direction of the Y axis motion.
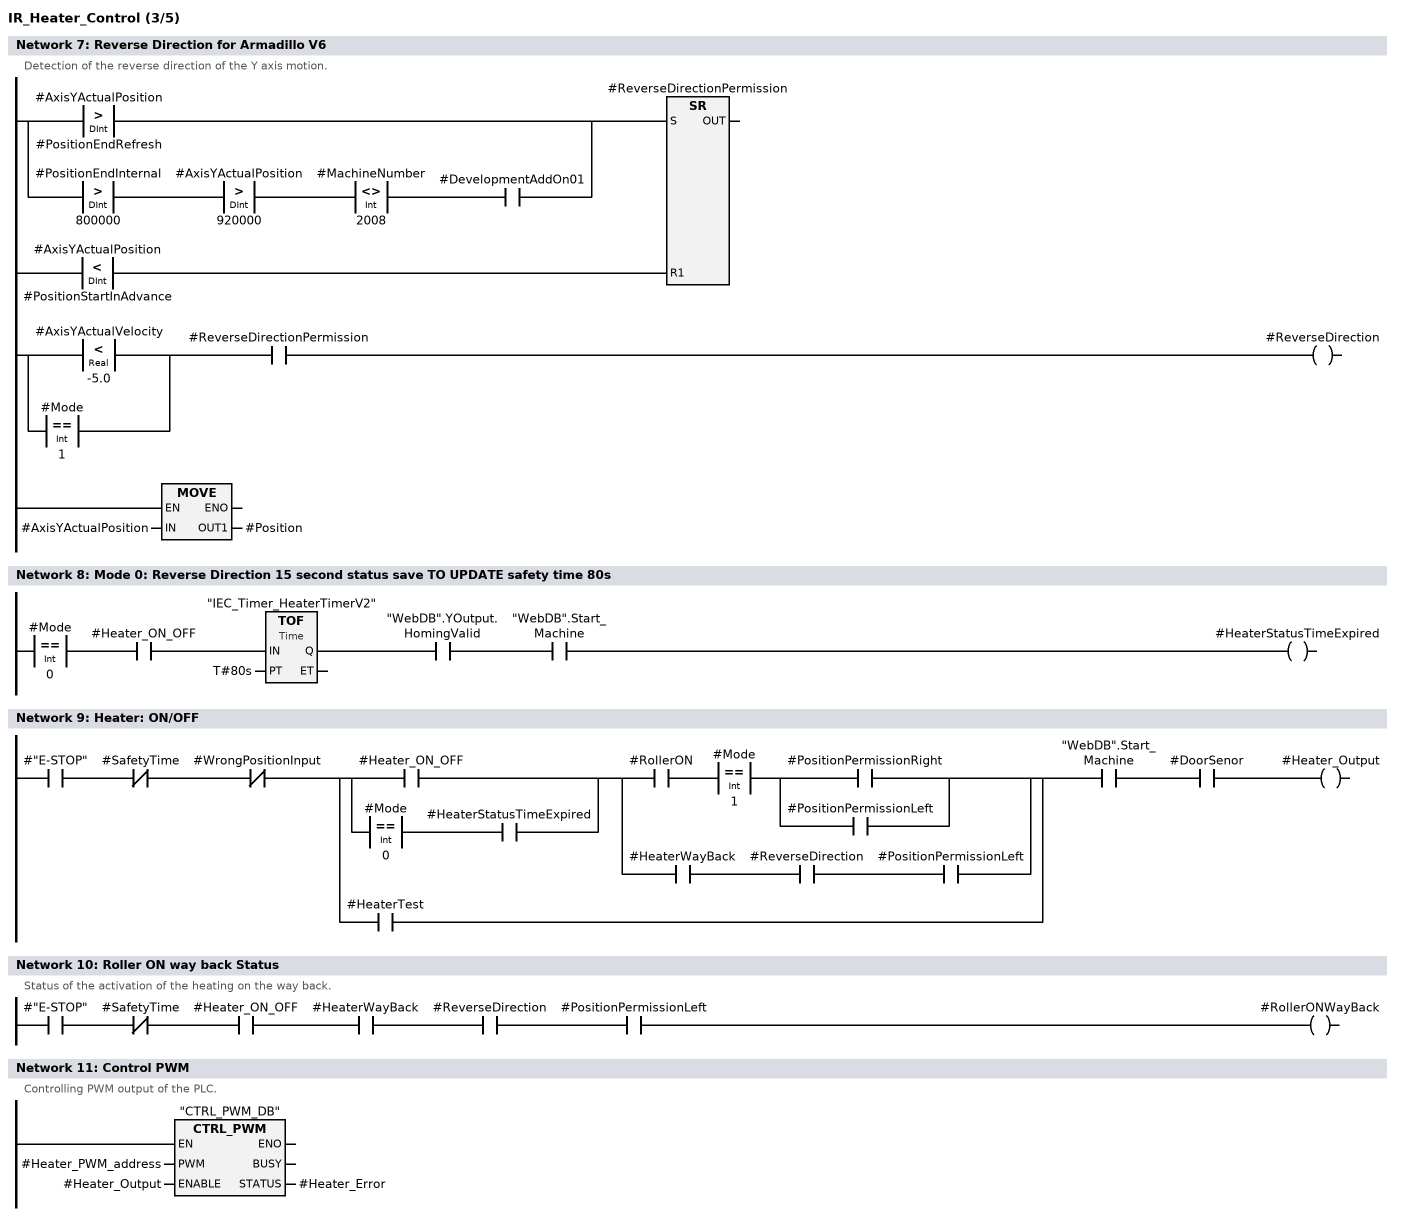
   RUNG wire#powerrail
      { S7_Templates := "SrcType := DInt" } GT_Contact(in1 := #AxisYActualPosition, in2 := #PositionEndRefresh)
      wire#w1
      S_SR(operand := #ReverseDirectionPermission, r1 := wire#w2)
   END_RUNG
   RUNG wire#powerrail
      { S7_Templates := "SrcType := DInt" } GT_Contact(in1 := #PositionEndInternal, in2 := 800000)
      { S7_Templates := "SrcType := DInt" } GT_Contact(in1 := #AxisYActualPosition, in2 := 920000)
      { S7_Templates := "SrcType := Int" } NE_Contact(in1 := #MachineNumber, in2 := 2008)
      Contact( #DevelopmentAddOn01 )
   END_RUNG wire#w1
   RUNG wire#powerrail
      { S7_Templates := "SrcType := DInt" } LT_Contact(in1 := #AxisYActualPosition, in2 := #PositionStartInAdvance)
   END_RUNG wire#w2
   RUNG wire#powerrail
      { S7_Templates := "SrcType := Real" } LT_Contact(in1 := #AxisYActualVelocity, in2 := -5.0)
      wire#w3
      Contact( #ReverseDirectionPermission )
      Coil( #ReverseDirection )
   END_RUNG
   RUNG wire#powerrail
      { S7_Templates := "SrcType := Int" } EQ_Contact(in1 := #Mode, in2 := 1)
   END_RUNG wire#w3
   RUNG wire#powerrail
      Move(in := #AxisYActualPosition, out1 => #Position)
   END_RUNG
   // the same network as SCL:
   IF (#AxisYActualPosition > #PositionEndRefresh) OR ((#PositionEndInternal > 800000) AND (#AxisYActualPosition > 920000) AND (#MachineNumber <> 2008) AND #DevelopmentAddOn01) THEN
       #ReverseDirectionPermission := TRUE;   // SR flip-flop
   END_IF;
   IF #AxisYActualPosition < #PositionStartInAdvance THEN #ReverseDirectionPermission := FALSE; END_IF;
   #ReverseDirection := ((#AxisYActualVelocity < (-5.0)) OR (#Mode = 1)) AND #ReverseDirectionPermission;
   #Position := #AxisYActualPosition;
END_REGION

REGION Network 8: Mode 0: Reverse Direction 15 second status save TO UPDATE safety time 80s
   RUNG wire#powerrail
      { S7_Templates := "SrcType := Int" } EQ_Contact(in1 := #Mode, in2 := 0)
      Contact( #Heater_ON_OFF )
      { S7_Templates := "time_type := Time" } "IEC_Timer_HeaterTimerV2".TOF(pt := T#80s, et =>)
      Contact( "WebDB".YOutput.HomingValid )
      Contact( "WebDB".Start_Machine )
      Coil( #HeaterStatusTimeExpired )
   END_RUNG
   // the same network as SCL:
   "IEC_Timer_HeaterTimerV2".TOF(IN := (#Mode = 0) AND #Heater_ON_OFF, PT := T#80s);
   #HeaterStatusTimeExpired := "IEC_Timer_HeaterTimerV2".Q AND "WebDB".YOutput.HomingValid AND "WebDB".Start_Machine;
END_REGION

REGION Network 9: Heater: ON/OFF
   RUNG wire#powerrail
      Contact( #"E-STOP" )
      I_Contact( #SafetyTime )
      I_Contact( #WrongPositionInput )
      wire#w1
      Contact( #Heater_ON_OFF )
      wire#w2
      Contact( #RollerON )
      { S7_Templates := "SrcType := Int" } EQ_Contact(in1 := #Mode, in2 := 1)
      wire#w3
      Contact( #PositionPermissionRight )
      wire#w4
      Contact( "WebDB".Start_Machine )
      Contact( #DoorSenor )
      Coil( #Heater_Output )
   END_RUNG
   RUNG wire#w1
      { S7_Templates := "SrcType := Int" } EQ_Contact(in1 := #Mode, in2 := 0)
      Contact( #HeaterStatusTimeExpired )
   END_RUNG wire#w2
   RUNG wire#w3
      Contact( #PositionPermissionLeft )
   END_RUNG wire#w4
   RUNG wire#w2
      Contact( #HeaterWayBack )
      Contact( #ReverseDirection )
      Contact( #PositionPermissionLeft )
   END_RUNG wire#w4
   RUNG wire#w1
      Contact( #HeaterTest )
   END_RUNG wire#w4
   // the same network as SCL:
   #Heater_Output := #"E-STOP" AND NOT #SafetyTime AND NOT #WrongPositionInput AND (((#Heater_ON_OFF OR ((#Mode = 0) AND #HeaterStatusTimeExpired)) AND ((#RollerON AND (#Mode = 1) AND (#PositionPermissionRight OR #PositionPermissionLeft)) OR (#HeaterWayBack AND #ReverseDirection AND #PositionPermissionLeft))) OR #HeaterTest) AND "WebDB".Start_Machine AND #DoorSenor;
END_REGION

REGION Network 10: Roller ON way back Status
   // Status of the activation of the heating on the way back.
   RUNG wire#powerrail
      Contact( #"E-STOP" )
      I_Contact( #SafetyTime )
      Contact( #Heater_ON_OFF )
      Contact( #HeaterWayBack )
      Contact( #ReverseDirection )
      Contact( #PositionPermissionLeft )
      Coil( #RollerONWayBack )
   END_RUNG
   // the same network as SCL:
   #RollerONWayBack := #"E-STOP" AND NOT #SafetyTime AND #Heater_ON_OFF AND #HeaterWayBack AND #ReverseDirection AND #PositionPermissionLeft;
END_REGION

REGION Network 11: Control PWM
   // Controlling PWM output of the PLC.
   RUNG wire#powerrail
      "CTRL_PWM_DB".CTRL_PWM(PWM := #Heater_PWM_address, ENABLE := #Heater_Output, BUSY =>, STATUS => #Heater_Error)
   END_RUNG
   // the same network as SCL:
   "CTRL_PWM_DB"(PWM := #Heater_PWM_address, ENABLE := #Heater_Output, STATUS => #Heater_Error);   // CTRL_PWM
END_REGION

REGION Network 12: Conversion
   // Conversion of the heater setpoint and limit.
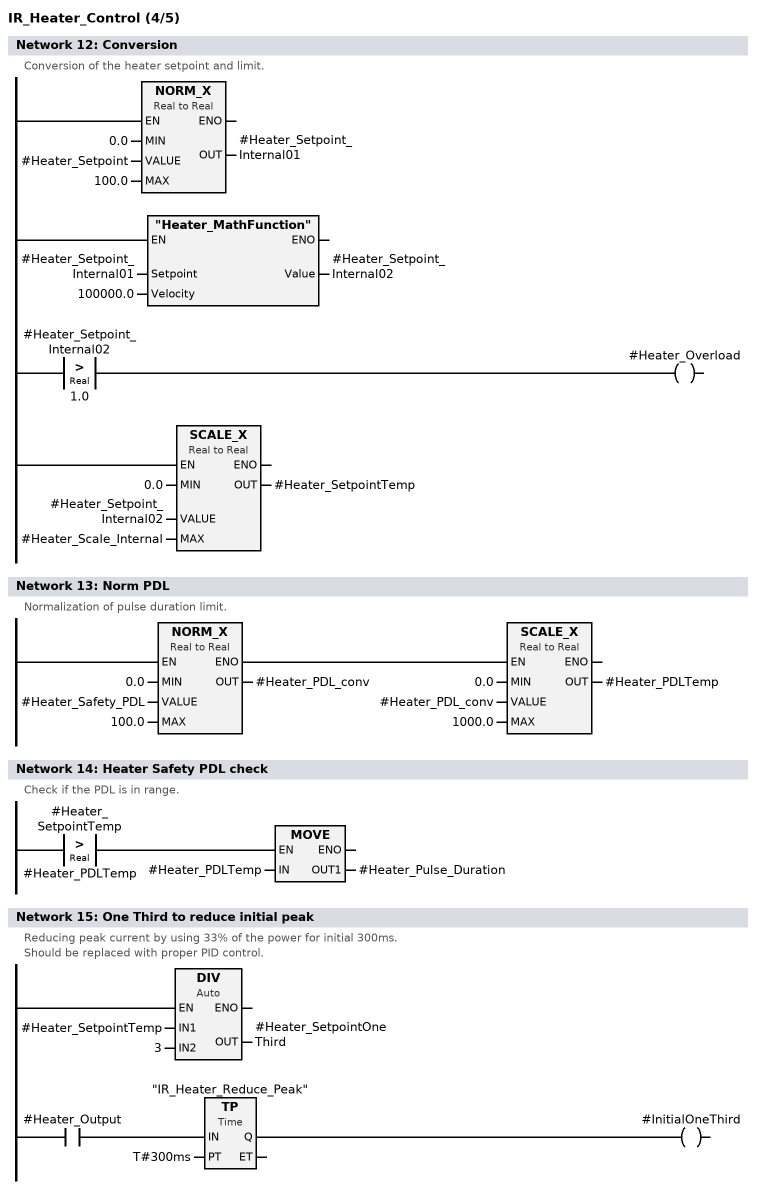
   RUNG wire#powerrail
      { S7_Templates := "[SrcType := Real, DestType := Real]" } Normalize(min := 0.0, value := #Heater_Setpoint, max := 100.0, out => #Heater_Setpoint_Internal01)
   END_RUNG
   RUNG wire#powerrail
      "Heater_MathFunction"(Setpoint := #Heater_Setpoint_Internal01, Velocity := 100000.0, Value => #Heater_Setpoint_Internal02)
   END_RUNG
   RUNG wire#powerrail
      { S7_Templates := "SrcType := Real" } GT_Contact(in1 := #Heater_Setpoint_Internal02, in2 := 1.0)
      Coil( #Heater_Overload )
   END_RUNG
   RUNG wire#powerrail
      { S7_Templates := "[SrcType := Real, DestType := Real]" } Scale(min := 0.0, value := #Heater_Setpoint_Internal02, max := #Heater_Scale_Internal, out => #Heater_SetpointTemp)
   END_RUNG
   // the same network as SCL:
   #Heater_Setpoint_Internal01 := NORM_X(MIN := 0.0, VALUE := #Heater_Setpoint, MAX := 100.0);
   "Heater_MathFunction"(Setpoint := #Heater_Setpoint_Internal01,
                         Velocity := 100000.0,
                         Value => #Heater_Setpoint_Internal02);
   #Heater_Overload := #Heater_Setpoint_Internal02 > 1.0;
   #Heater_SetpointTemp := SCALE_X(MIN := 0.0, VALUE := #Heater_Setpoint_Internal02, MAX := #Heater_Scale_Internal);
END_REGION

REGION Network 13: Norm PDL
   // Normalization of pulse duration limit.
   RUNG wire#powerrail
      { S7_Templates := "[SrcType := Real, DestType := Real]" } Normalize(min := 0.0, value := #Heater_Safety_PDL, max := 100.0, out => #Heater_PDL_conv)
      { S7_Templates := "[SrcType := Real, DestType := Real]" } Scale(min := 0.0, value := #Heater_PDL_conv, max := 1000.0, out => #Heater_PDLTemp)
   END_RUNG
   // the same network as SCL:
   #Heater_PDL_conv := NORM_X(MIN := 0.0, VALUE := #Heater_Safety_PDL, MAX := 100.0);
   #Heater_PDLTemp := SCALE_X(MIN := 0.0, VALUE := #Heater_PDL_conv, MAX := 1000.0);
END_REGION

REGION Network 14: Heater Safety PDL check
   // Check if the PDL is in range.
   RUNG wire#powerrail
      { S7_Templates := "SrcType := Real" } GT_Contact(in1 := #Heater_SetpointTemp, in2 := #Heater_PDLTemp)
      Move(in := #Heater_PDLTemp, out1 => #Heater_Pulse_Duration)
   END_RUNG
   // the same network as SCL:
   IF #Heater_SetpointTemp > #Heater_PDLTemp THEN #Heater_Pulse_Duration := #Heater_PDLTemp; END_IF;
END_REGION

REGION Network 15: One Third to reduce initial peak
   // Reducing peak current by using 33% of the power for initial 300ms.
   // 
   // Should be replaced with proper PID control.
   RUNG wire#powerrail
      Div(in1 := #Heater_SetpointTemp, in2 := 3, out => #Heater_SetpointOneThird)
   END_RUNG
   RUNG wire#powerrail
      Contact( #Heater_Output )
      { S7_Templates := "time_type := Time" } "IR_Heater_Reduce_Peak".TP(pt := T#300ms, et =>)
      Coil( #InitialOneThird )
   END_RUNG
   // the same network as SCL:
   #Heater_SetpointOneThird := #Heater_SetpointTemp / 3;
   "IR_Heater_Reduce_Peak".TP(IN := #Heater_Output, PT := T#300ms);
   #InitialOneThird := "IR_Heater_Reduce_Peak".Q;
END_REGION

REGION Network 16: Move
   // Moving heating parameters.
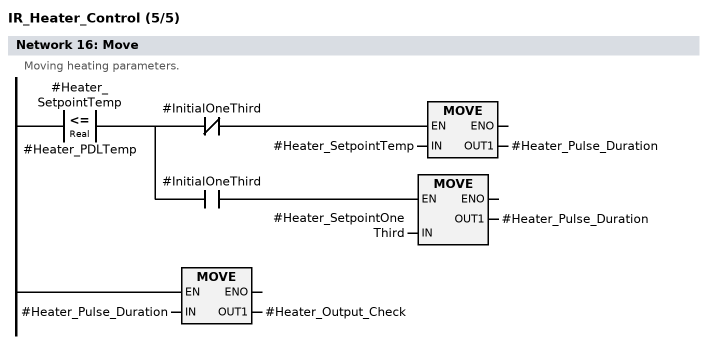
   RUNG wire#powerrail
      { S7_Templates := "SrcType := Real" } LE_Contact(in1 := #Heater_SetpointTemp, in2 := #Heater_PDLTemp)
      wire#w1
      I_Contact( #InitialOneThird )
      Move(in := #Heater_SetpointTemp, out1 => #Heater_Pulse_Duration)
   END_RUNG
   RUNG wire#w1
      Contact( #InitialOneThird )
      Move(in := #Heater_SetpointOneThird, out1 => #Heater_Pulse_Duration)
   END_RUNG
   RUNG wire#powerrail
      Move(in := #Heater_Pulse_Duration, out1 => #Heater_Output_Check)
   END_RUNG
   // the same network as SCL:
   #_w1 := #Heater_SetpointTemp <= #Heater_PDLTemp;
   IF #_w1 AND NOT #InitialOneThird THEN #Heater_Pulse_Duration := #Heater_SetpointTemp; END_IF;
   IF #_w1 AND #InitialOneThird THEN #Heater_Pulse_Duration := #Heater_SetpointOneThird; END_IF;
   #Heater_Output_Check := #Heater_Pulse_Duration;
END_REGION
END_FUNCTION_BLOCK

FUNCTION "Heater_MathFunction" : Void
{ S7_Optimized_Access := 'TRUE' }
VERSION : 0.1
   VAR_INPUT 
      Setpoint : Real;
      Velocity : Real;
   END_VAR

   VAR_OUTPUT 
      Value : Real;
   END_VAR


BEGIN
	// Math Function Implementation for IR Heater
	#Value := (#Velocity / 100000) * #Setpoint;
	
END_FUNCTION

FUNCTION_BLOCK "LoadCell"   // FB7, LAD
TITLE = Description:
{ S7_Optimized_Access := 'TRUE' }
VERSION : 0.1
// Old control block - should be checked described.
   VAR_INPUT
      MinValue : UInt := 0;
      MaxValue : UInt := 27648;
      ILoadCell : UInt;
      Const_V : UInt := 10;
      Const_SubWeight : Real := 0.629;
      Const_Kg : UInt := 13970;
   END_VAR
   VAR_OUTPUT
      OWeight : UInt;
   END_VAR
   VAR_TEMP
      NormVal : Real;
      ScalVal : Real;
      SubVal : Real;
      MulVal : Real;
   END_VAR
BEGIN

REGION Network 1
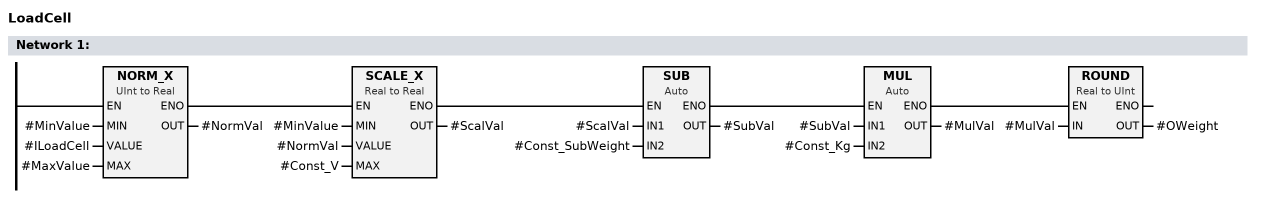
   RUNG wire#powerrail
      { S7_Templates := "[SrcType := UInt, DestType := Real]" } Normalize(min := #MinValue, value := #ILoadCell, max := #MaxValue, out => #NormVal)
      { S7_Templates := "[SrcType := Real, DestType := Real]" } Scale(min := #MinValue, value := #NormVal, max := #Const_V, out => #ScalVal)
      Sub(in1 := #ScalVal, in2 := #Const_SubWeight, out => #SubVal)
      Mul(in1 := #SubVal, in2 := #Const_Kg, out => #MulVal)
      { S7_Templates := "[SrcType := Real, DestType := UInt]" } Round(in := #MulVal, out => #OWeight)
   END_RUNG
   // the same network as SCL:
   #NormVal := NORM_X(MIN := #MinValue, VALUE := #ILoadCell, MAX := #MaxValue);
   #ScalVal := SCALE_X(MIN := #MinValue, VALUE := #NormVal, MAX := #Const_V);
   #SubVal := #ScalVal - #Const_SubWeight;
   #MulVal := #SubVal * #Const_Kg;
   #OWeight := ROUND(#MulVal);
END_REGION
END_FUNCTION_BLOCK

FUNCTION_BLOCK "LED_Behavior"   // FB11, LAD
TITLE = Description:
{ S7_Optimized_Access := 'TRUE' }
VERSION : 0.1
// Old control block - should be checked and described.
   VAR_INPUT
      RED : Bool;
      GREEN : Bool;
      RED_BLINK : Bool;
      GREEN_BLINK : Bool;
      RED_GREEN_BLINK : Bool;
   END_VAR
   VAR_OUTPUT
      LED_1_Output : Bool;
      LED_2_Output : Bool;
   END_VAR
   VAR
      Red_Blink_Output : Bool;
      Green_Blink_Output : Bool;
      "Red/Green_Blink_Output" : Bool;
      Red_Blink_M : Bool;
      Red_Blink_S : Bool;
      Green_Blink_M : Bool;
      Green_Blink_S : Bool;
      Reset_Red_Blink : Bool;
      Reset_Green_Blink : Bool;
      Reset_RED_GREEN_Blink : Bool;
      RG_Blink_M : Bool;
      RG_Blink_S : Bool;
   END_VAR
BEGIN

REGION Network 1: Output 1 Color 1=RED 0=GREEN
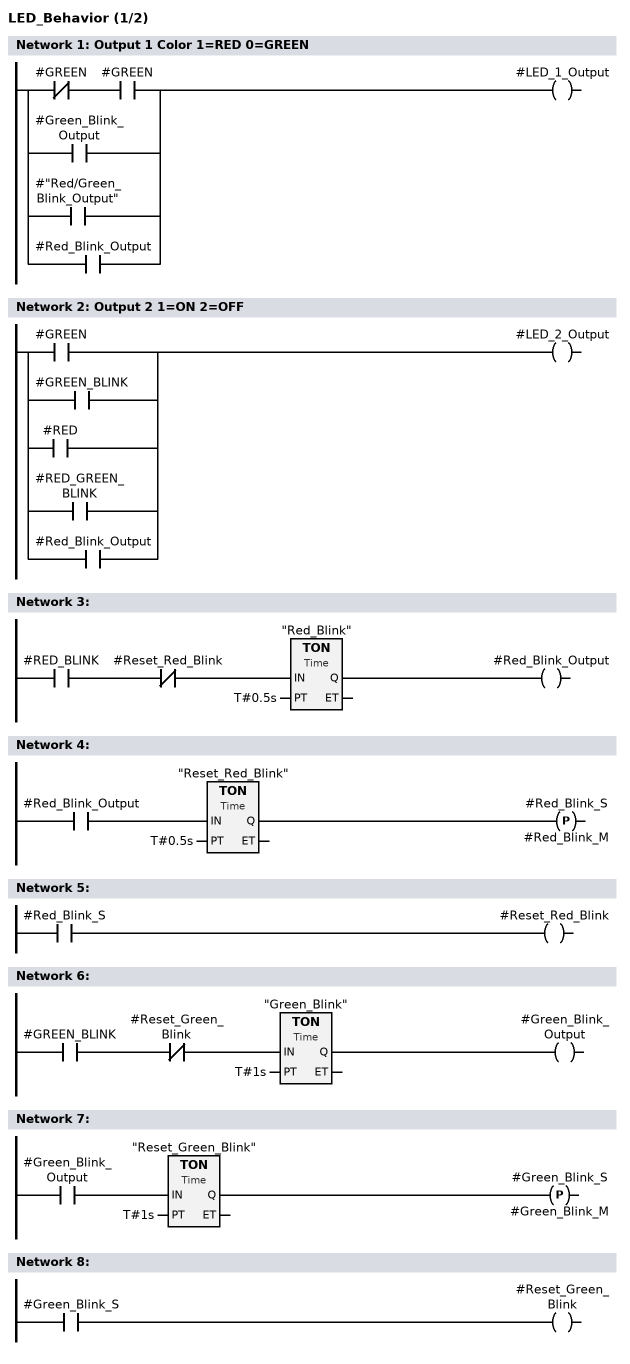
   RUNG wire#powerrail
      I_Contact( #GREEN )
      Contact( #GREEN )
      wire#w1
      Coil( #LED_1_Output )
   END_RUNG
   RUNG wire#powerrail
      Contact( #Green_Blink_Output )
   END_RUNG wire#w1
   RUNG wire#powerrail
      Contact( #"Red/Green_Blink_Output" )
   END_RUNG wire#w1
   RUNG wire#powerrail
      Contact( #Red_Blink_Output )
   END_RUNG wire#w1
   // the same network as SCL:
   #LED_1_Output := (NOT #GREEN AND #GREEN) OR #Green_Blink_Output OR #"Red/Green_Blink_Output" OR #Red_Blink_Output;
END_REGION

REGION Network 2: Output 2 1=ON 2=OFF
   RUNG wire#powerrail
      Contact( #GREEN )
      wire#w1
      Coil( #LED_2_Output )
   END_RUNG
   RUNG wire#powerrail
      Contact( #GREEN_BLINK )
   END_RUNG wire#w1
   RUNG wire#powerrail
      Contact( #RED )
   END_RUNG wire#w1
   RUNG wire#powerrail
      Contact( #RED_GREEN_BLINK )
   END_RUNG wire#w1
   RUNG wire#powerrail
      Contact( #Red_Blink_Output )
   END_RUNG wire#w1
   // the same network as SCL:
   #LED_2_Output := #GREEN OR #GREEN_BLINK OR #RED OR #RED_GREEN_BLINK OR #Red_Blink_Output;
END_REGION

REGION Network 3
   RUNG wire#powerrail
      Contact( #RED_BLINK )
      I_Contact( #Reset_Red_Blink )
      { S7_Templates := "time_type := Time" } "Red_Blink".TON(pt := T#0.5s, et =>)
      Coil( #Red_Blink_Output )
   END_RUNG
   // the same network as SCL:
   "Red_Blink".TON(IN := #RED_BLINK AND NOT #Reset_Red_Blink, PT := T#0.5s);
   #Red_Blink_Output := "Red_Blink".Q;
END_REGION

REGION Network 4
   "Reset_Red_Blink".TON(IN := #Red_Blink_Output, PT := T#0.5s);
   #Red_Blink_S := "Reset_Red_Blink".Q AND NOT #Red_Blink_M;   // rising edge
   #Red_Blink_M := "Reset_Red_Blink".Q;
END_REGION

REGION Network 5
   RUNG wire#powerrail
      Contact( #Red_Blink_S )
      Coil( #Reset_Red_Blink )
   END_RUNG
   // the same network as SCL:
   #Reset_Red_Blink := #Red_Blink_S;
END_REGION

REGION Network 6
   RUNG wire#powerrail
      Contact( #GREEN_BLINK )
      I_Contact( #Reset_Green_Blink )
      { S7_Templates := "time_type := Time" } "Green_Blink".TON(pt := T#1s, et =>)
      Coil( #Green_Blink_Output )
   END_RUNG
   // the same network as SCL:
   "Green_Blink".TON(IN := #GREEN_BLINK AND NOT #Reset_Green_Blink, PT := T#1s);
   #Green_Blink_Output := "Green_Blink".Q;
END_REGION

REGION Network 7
   "Reset_Green_Blink".TON(IN := #Green_Blink_Output, PT := T#1s);
   #Green_Blink_S := "Reset_Green_Blink".Q AND NOT #Green_Blink_M;   // rising edge
   #Green_Blink_M := "Reset_Green_Blink".Q;
END_REGION

REGION Network 8
   RUNG wire#powerrail
      Contact( #Green_Blink_S )
      Coil( #Reset_Green_Blink )
   END_RUNG
   // the same network as SCL:
   #Reset_Green_Blink := #Green_Blink_S;
END_REGION

REGION Network 9
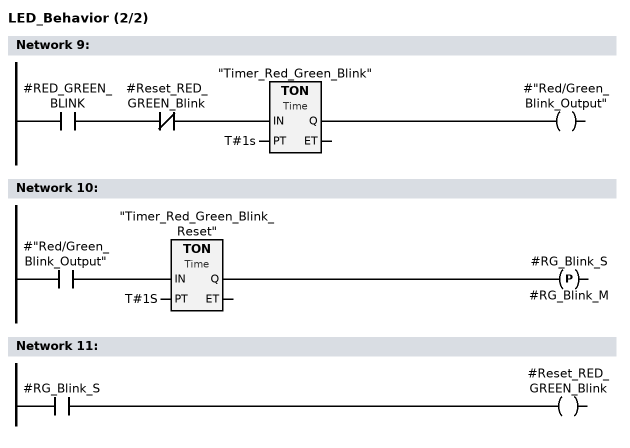
   RUNG wire#powerrail
      Contact( #RED_GREEN_BLINK )
      I_Contact( #Reset_RED_GREEN_Blink )
      { S7_Templates := "time_type := Time" } "Timer_Red_Green_Blink".TON(pt := T#1s, et =>)
      Coil( #"Red/Green_Blink_Output" )
   END_RUNG
   // the same network as SCL:
   "Timer_Red_Green_Blink".TON(IN := #RED_GREEN_BLINK AND NOT #Reset_RED_GREEN_Blink, PT := T#1s);
   #"Red/Green_Blink_Output" := "Timer_Red_Green_Blink".Q;
END_REGION

REGION Network 10
   "Timer_Red_Green_Blink_Reset".TON(IN := #"Red/Green_Blink_Output", PT := T#1S);
   #RG_Blink_S := "Timer_Red_Green_Blink_Reset".Q AND NOT #RG_Blink_M;   // rising edge
   #RG_Blink_M := "Timer_Red_Green_Blink_Reset".Q;
END_REGION

REGION Network 11
   RUNG wire#powerrail
      Contact( #RG_Blink_S )
      Coil( #Reset_RED_GREEN_Blink )
   END_RUNG
   // the same network as SCL:
   #Reset_RED_GREEN_Blink := #RG_Blink_S;
END_REGION
END_FUNCTION_BLOCK

FUNCTION_BLOCK "Capping_Station"   // FB1, LAD
TITLE = Description
{ S7_Optimized_Access := 'TRUE' }
VERSION : 0.1
// How to control and set capping station:
// 1) Start the machine
// 2) Use jog pos/neg in the capping station data block to rotate motor to read max and min value: ReadSensorMax and Read SensorMin. Based on these values update "SensorPosValMax..." and "SensorPosValMin..."
// 3) Move capping station using "MovingUP" and "MovingDOWN". The mechanism should stop top or bottom and confirm it with the change of the status "CSPositionUP" and "CSPositionDOWN". If it is constantly moving, it means that the value was not reached (too low for SensorPosValMin or too high for "SensorPosValMax").
// 
// IMPORTANT:
// - assembly of the mechanism needs to be the same, especially the position of the sensor
// - power supply for the sensor should be set to the exact voltage (5V) to provide repeteable readings
// 
// Things to implement:
// - Change sensor for limit switch
// - Improve mechanical design
// 
// E-STOP - always check!
   VAR_INPUT
      ESTOP : Bool;
      SerialNumber : Int;
      CappingOption : Int;   // Send 1 to skip capping station
      MachineStart : Bool;
      CappingSensor : UInt;
      JogPOS : Bool;
      JogNEG : Bool;
      MoveRel : Bool;
      AxisXNotMoving : Bool;
      AxisYNotMoving : Bool;
      DoorSensor : Bool;
   END_VAR
   VAR_OUTPUT
      MovingUP : Bool;
      MovingDOWN : Bool;
      CSPositionUP : Bool;
      CSPositionDOWN : Bool;
      CSXYMotionLock : Bool;
      CappingPosition : UInt;
      MaintenanceNeeded : Bool;
   END_VAR
   VAR_IN_OUT
      CSMoveUP : Bool;
      CSMoveDOWN : Bool;
   END_VAR
   VAR
      MotionLockInternal : Bool;
      TimeSafety : Bool;
      SensorConversion : Real;
      SensorPosValMaxTrigger : UInt;
      SensorPosValMinTrigger : UInt;
      ReadSensorMax : UInt;   // Use jogging to read initial limit values
      ReadSensorMin : UInt := 10000;   // Use jogging to read initial limit values
      CountSinceON : DInt;
   END_VAR
   VAR RETAIN
      CountSinceNEW : DInt;
   END_VAR
   VAR
      MaintenanceMotionLockDisabled : Bool := true;
      SensorPosValMin : UInt;   // 0; 14000; Machine 2009: 9000
      SensorPosValMax : UInt;   // 6000; 21000; Machine 2009: 24500
      ScaleRangeMin : UInt;   // 2009: 26000; 2008 20000;
      ScaleRangeMax : UInt;   // 2009: 12000; 2008 4200;
   END_VAR
   VAR_TEMP
      JoggingPOSInternal : Bool;
      JoggingNEGInternal : Bool;
      CSPositionUPInternal : Bool;
      CSPositionDOWNInternal : Bool;
      MovingPermission : Bool;
   END_VAR
   VAR CONSTANT
      SensorPosValMax2008 : UInt := 15000;
      SensorPosValMax2009 : UInt := 24500;   // Armadillo 2009
      SensorPosValMax2010 : UInt := 17000;   // Armadillo 2010
      SensorPosValMax2011 : UInt := 13000;
      SensorPosValMax2012 : UInt := 14000;
      SensorPosValMin2008 : UInt := 5300;
      SensorPosValMin2009 : UInt := 9000;   // Armadillo 2009
      SensorPosValMin2010 : UInt := 4300;   // Armadillo 2010
      SensorPosValMin2011 : UInt := 4300;
      SensorPosValMin2012 : UInt := 4300;
      SensorPosTopMargin : UInt := 2000;   // 2000
      SensorPosBottomMargin : UInt := 2000;   // 2000
      ScaleRangeMax2008 : UInt := 18000;
      ScaleRangeMax2009 : UInt := 26000;
      ScaleRangeMax2010 : UInt := 18000;
      ScaleRangeMax2011 : UInt := 18000;
      ScaleRangeMax2012 : UInt := 18000;
      ScaleRangeMin2008 : UInt := 8000;
      ScaleRangeMin2009 : UInt := 8000;
      ScaleRangeMin2010 : UInt := 4200;
      ScaleRangeMin2011 : UInt := 8000;
      ScaleRangeMin2012 : UInt := 8000;
      MoveLength : DInt := 10000;   // microns
      MovementVelocity : Real := 90.0;   // 90
   END_VAR
   VAR_TEMP   // added for the SCL form of the ladder/FBD networks
      _w1 : Bool;
   END_VAR
BEGIN

REGION Network 1: Limit settings for different machines
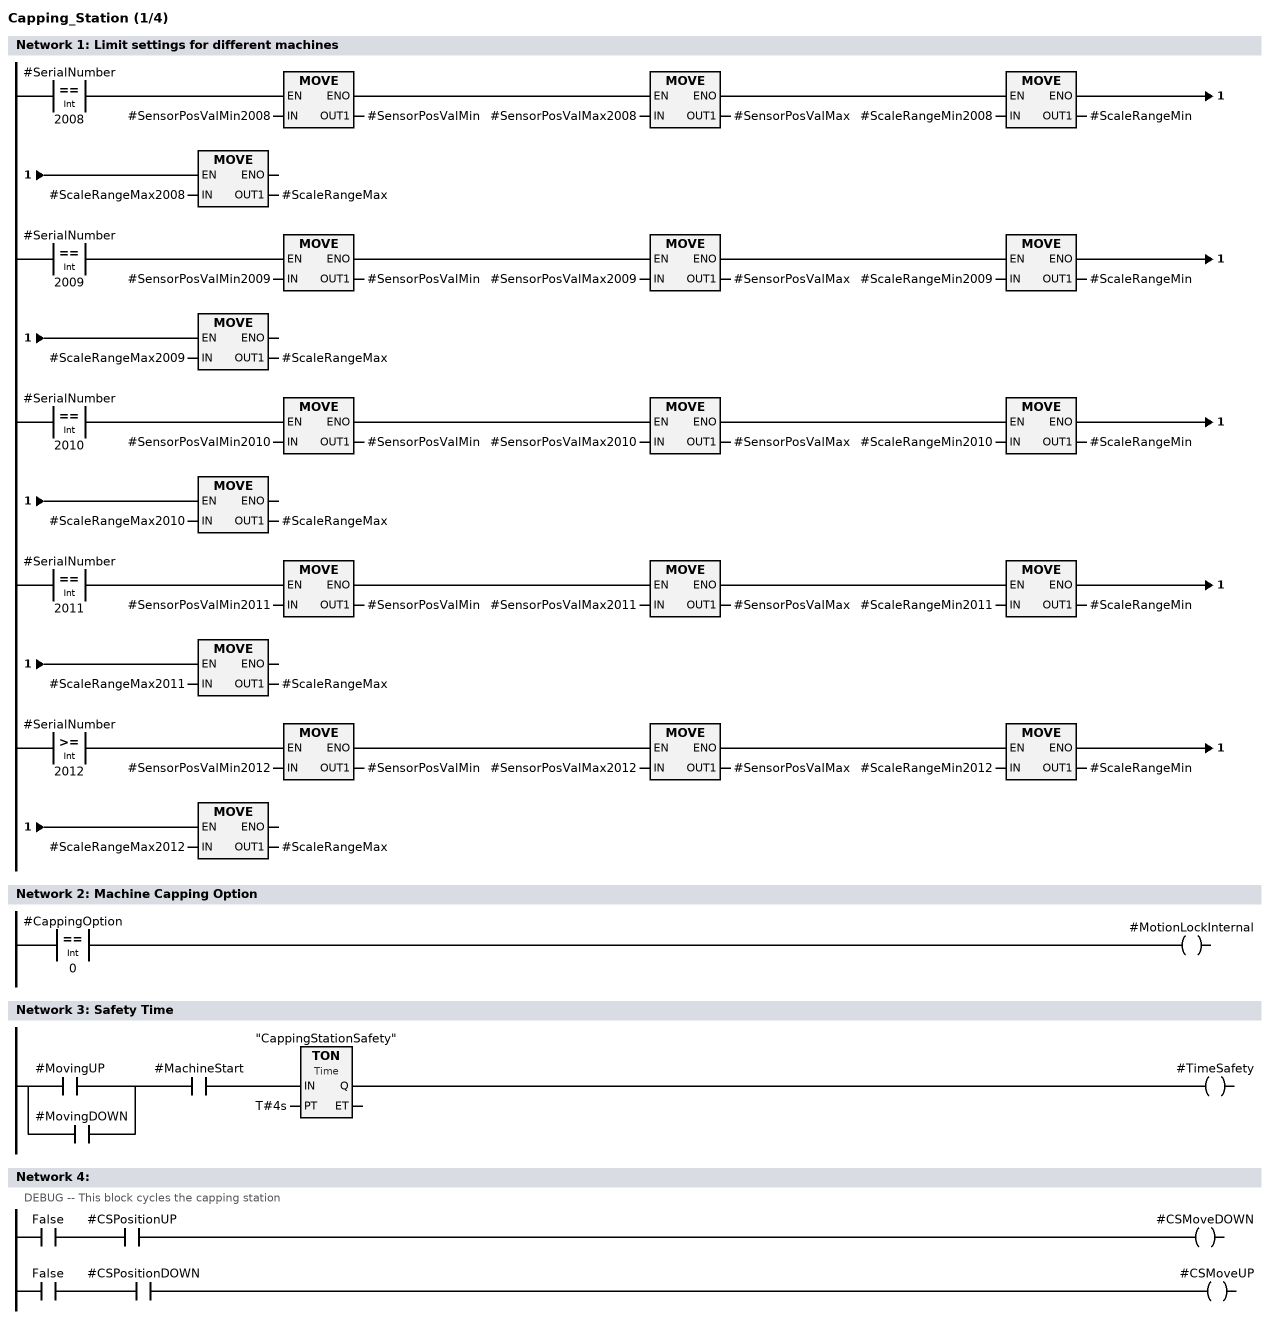
   RUNG wire#powerrail
      { S7_Templates := "SrcType := Int" } EQ_Contact(in1 := #SerialNumber, in2 := 2008)
      Move(in := #SensorPosValMin2008, out1 => #SensorPosValMin)
      Move(in := #SensorPosValMax2008, out1 => #SensorPosValMax)
      Move(in := #ScaleRangeMin2008, out1 => #ScaleRangeMin)
      Move(in := #ScaleRangeMax2008, out1 => #ScaleRangeMax)
   END_RUNG
   RUNG wire#powerrail
      { S7_Templates := "SrcType := Int" } EQ_Contact(in1 := #SerialNumber, in2 := 2009)
      Move(in := #SensorPosValMin2009, out1 => #SensorPosValMin)
      Move(in := #SensorPosValMax2009, out1 => #SensorPosValMax)
      Move(in := #ScaleRangeMin2009, out1 => #ScaleRangeMin)
      Move(in := #ScaleRangeMax2009, out1 => #ScaleRangeMax)
   END_RUNG
   RUNG wire#powerrail
      { S7_Templates := "SrcType := Int" } EQ_Contact(in1 := #SerialNumber, in2 := 2010)
      Move(in := #SensorPosValMin2010, out1 => #SensorPosValMin)
      Move(in := #SensorPosValMax2010, out1 => #SensorPosValMax)
      Move(in := #ScaleRangeMin2010, out1 => #ScaleRangeMin)
      Move(in := #ScaleRangeMax2010, out1 => #ScaleRangeMax)
   END_RUNG
   RUNG wire#powerrail
      { S7_Templates := "SrcType := Int" } EQ_Contact(in1 := #SerialNumber, in2 := 2011)
      Move(in := #SensorPosValMin2011, out1 => #SensorPosValMin)
      Move(in := #SensorPosValMax2011, out1 => #SensorPosValMax)
      Move(in := #ScaleRangeMin2011, out1 => #ScaleRangeMin)
      Move(in := #ScaleRangeMax2011, out1 => #ScaleRangeMax)
   END_RUNG
   RUNG wire#powerrail
      { S7_Templates := "SrcType := Int" } GE_Contact(in1 := #SerialNumber, in2 := 2012)
      Move(in := #SensorPosValMin2012, out1 => #SensorPosValMin)
      Move(in := #SensorPosValMax2012, out1 => #SensorPosValMax)
      Move(in := #ScaleRangeMin2012, out1 => #ScaleRangeMin)
      Move(in := #ScaleRangeMax2012, out1 => #ScaleRangeMax)
   END_RUNG
   // the same network as SCL:
   IF #SerialNumber = 2008 THEN
       #SensorPosValMin := #SensorPosValMin2008;
       #SensorPosValMax := #SensorPosValMax2008;
       #ScaleRangeMin := #ScaleRangeMin2008;
       #ScaleRangeMax := #ScaleRangeMax2008;
   END_IF;
   IF #SerialNumber = 2009 THEN
       #SensorPosValMin := #SensorPosValMin2009;
       #SensorPosValMax := #SensorPosValMax2009;
       #ScaleRangeMin := #ScaleRangeMin2009;
       #ScaleRangeMax := #ScaleRangeMax2009;
   END_IF;
   IF #SerialNumber = 2010 THEN
       #SensorPosValMin := #SensorPosValMin2010;
       #SensorPosValMax := #SensorPosValMax2010;
       #ScaleRangeMin := #ScaleRangeMin2010;
       #ScaleRangeMax := #ScaleRangeMax2010;
   END_IF;
   IF #SerialNumber = 2011 THEN
       #SensorPosValMin := #SensorPosValMin2011;
       #SensorPosValMax := #SensorPosValMax2011;
       #ScaleRangeMin := #ScaleRangeMin2011;
       #ScaleRangeMax := #ScaleRangeMax2011;
   END_IF;
   IF #SerialNumber >= 2012 THEN
       #SensorPosValMin := #SensorPosValMin2012;
       #SensorPosValMax := #SensorPosValMax2012;
       #ScaleRangeMin := #ScaleRangeMin2012;
       #ScaleRangeMax := #ScaleRangeMax2012;
   END_IF;
END_REGION

REGION Network 2: Machine Capping Option
   RUNG wire#powerrail
      { S7_Templates := "SrcType := Int" } EQ_Contact(in1 := #CappingOption, in2 := 0)
      Coil( #MotionLockInternal )
   END_RUNG
   // the same network as SCL:
   #MotionLockInternal := #CappingOption = 0;
END_REGION

REGION Network 3: Safety Time
   RUNG wire#powerrail
      Contact( #MovingUP )
      wire#w1
      Contact( #MachineStart )
      { S7_Templates := "time_type := Time" } "CappingStationSafety".TON(pt := T#4s, et =>)
      Coil( #TimeSafety )
   END_RUNG
   RUNG wire#powerrail
      Contact( #MovingDOWN )
   END_RUNG wire#w1
   // the same network as SCL:
   "CappingStationSafety".TON(IN := (#MovingUP OR #MovingDOWN) AND #MachineStart, PT := T#4s);
   #TimeSafety := "CappingStationSafety".Q;
END_REGION

REGION Network 4
   // DEBUG -- This block cycles the capping station
   RUNG wire#powerrail
      Contact( False )
      Contact( #CSPositionUP )
      Coil( #CSMoveDOWN )
   END_RUNG
   RUNG wire#powerrail
      Contact( False )
      Contact( #CSPositionDOWN )
      Coil( #CSMoveUP )
   END_RUNG
   // the same network as SCL:
   #CSMoveDOWN := False AND #CSPositionUP;
   #CSMoveUP := False AND #CSPositionDOWN;
END_REGION

REGION Network 5: Read Sensor Range
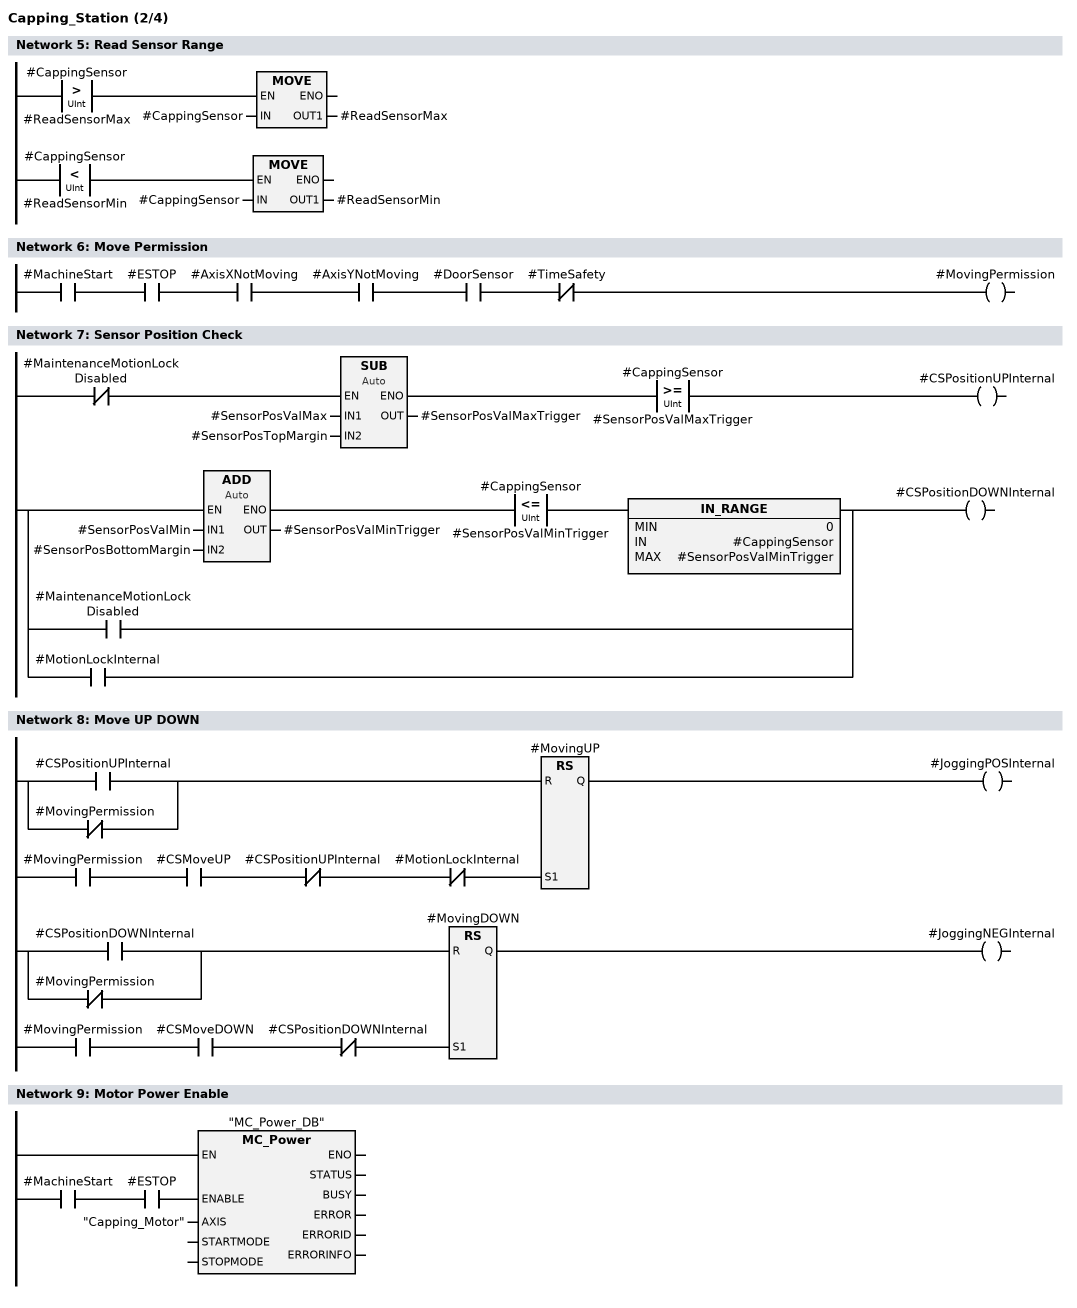
   RUNG wire#powerrail
      { S7_Templates := "SrcType := UInt" } GT_Contact(in1 := #CappingSensor, in2 := #ReadSensorMax)
      Move(in := #CappingSensor, out1 => #ReadSensorMax)
   END_RUNG
   RUNG wire#powerrail
      { S7_Templates := "SrcType := UInt" } LT_Contact(in1 := #CappingSensor, in2 := #ReadSensorMin)
      Move(in := #CappingSensor, out1 => #ReadSensorMin)
   END_RUNG
   // the same network as SCL:
   IF #CappingSensor > #ReadSensorMax THEN #ReadSensorMax := #CappingSensor; END_IF;
   IF #CappingSensor < #ReadSensorMin THEN #ReadSensorMin := #CappingSensor; END_IF;
END_REGION

REGION Network 6: Move Permission
   RUNG wire#powerrail
      Contact( #MachineStart )
      Contact( #ESTOP )
      Contact( #AxisXNotMoving )
      Contact( #AxisYNotMoving )
      Contact( #DoorSensor )
      I_Contact( #TimeSafety )
      Coil( #MovingPermission )
   END_RUNG
   // the same network as SCL:
   #MovingPermission := #MachineStart AND #ESTOP AND #AxisXNotMoving AND #AxisYNotMoving AND #DoorSensor AND NOT #TimeSafety;
END_REGION

REGION Network 7: Sensor Position Check
   RUNG wire#powerrail
      I_Contact( #MaintenanceMotionLockDisabled )
      Sub(in1 := #SensorPosValMax, in2 := #SensorPosTopMargin, out => #SensorPosValMaxTrigger)
      { S7_Templates := "SrcType := UInt" } GE_Contact(in1 := #CappingSensor, in2 := #SensorPosValMaxTrigger)
      Coil( #CSPositionUPInternal )
   END_RUNG
   RUNG wire#powerrail
      Add(in1 := #SensorPosValMin, in2 := #SensorPosBottomMargin, out => #SensorPosValMinTrigger)
      { S7_Templates := "SrcType := UInt" } LE_Contact(in1 := #CappingSensor, in2 := #SensorPosValMinTrigger)
      { S7_Templates := "SrcType := UInt" } InRange(min := 0, in := #CappingSensor, max := #SensorPosValMinTrigger)
      wire#w1
      Coil( #CSPositionDOWNInternal )
   END_RUNG
   RUNG wire#powerrail
      Contact( #MaintenanceMotionLockDisabled )
   END_RUNG wire#w1
   RUNG wire#powerrail
      Contact( #MotionLockInternal )
   END_RUNG wire#w1
   // the same network as SCL:
   #_w1 := NOT #MaintenanceMotionLockDisabled;
   IF #_w1 THEN #SensorPosValMaxTrigger := #SensorPosValMax - #SensorPosTopMargin; END_IF;
   #CSPositionUPInternal := #_w1 AND (#CappingSensor >= #SensorPosValMaxTrigger);
   #SensorPosValMinTrigger := #SensorPosValMin + #SensorPosBottomMargin;
   #CSPositionDOWNInternal := ((#CappingSensor <= #SensorPosValMinTrigger) AND (0 <= #CappingSensor) AND (#CappingSensor <= #SensorPosValMinTrigger)) OR #MaintenanceMotionLockDisabled OR #MotionLockInternal;
END_REGION

REGION Network 8: Move UP DOWN
   RUNG wire#powerrail
      Contact( #CSPositionUPInternal )
      wire#w1
      S_RS(operand := #MovingUP, s1 := wire#w2)
      Coil( #JoggingPOSInternal )
   END_RUNG
   RUNG wire#powerrail
      I_Contact( #MovingPermission )
   END_RUNG wire#w1
   RUNG wire#powerrail
      Contact( #MovingPermission )
      Contact( #CSMoveUP )
      I_Contact( #CSPositionUPInternal )
      I_Contact( #MotionLockInternal )
   END_RUNG wire#w2
   RUNG wire#powerrail
      Contact( #CSPositionDOWNInternal )
      wire#w3
      S_RS(operand := #MovingDOWN, s1 := wire#w4)
      Coil( #JoggingNEGInternal )
   END_RUNG
   RUNG wire#powerrail
      I_Contact( #MovingPermission )
   END_RUNG wire#w3
   RUNG wire#powerrail
      Contact( #MovingPermission )
      Contact( #CSMoveDOWN )
      I_Contact( #CSPositionDOWNInternal )
   END_RUNG wire#w4
   // the same network as SCL:
   IF #CSPositionUPInternal OR NOT #MovingPermission THEN
       #MovingUP := FALSE;   // RS flip-flop
   END_IF;
   IF #MovingPermission AND #CSMoveUP AND NOT #CSPositionUPInternal AND NOT #MotionLockInternal THEN
       #MovingUP := TRUE;
   END_IF;
   #JoggingPOSInternal := #MovingUP;
   IF #CSPositionDOWNInternal OR NOT #MovingPermission THEN
       #MovingDOWN := FALSE;   // RS flip-flop
   END_IF;
   IF #MovingPermission AND #CSMoveDOWN AND NOT #CSPositionDOWNInternal THEN #MovingDOWN := TRUE; END_IF;
   #JoggingNEGInternal := #MovingDOWN;
END_REGION

REGION Network 9: Motor Power Enable
   RUNG wire#powerrail
      "MC_Power_DB".MC_Power(Enable := wire#w1, Axis := "Capping_Motor", StartMode :=, StopMode :=, Status =>, Busy =>, Error =>, ErrorID =>, ErrorInfo =>)
   END_RUNG
   RUNG wire#powerrail
      Contact( #MachineStart )
      Contact( #ESTOP )
   END_RUNG wire#w1
   // the same network as SCL:
   "MC_Power_DB"(Enable := #MachineStart AND #ESTOP, Axis := "Capping_Motor");   // MC_Power
END_REGION

REGION Network 10: Move Jog
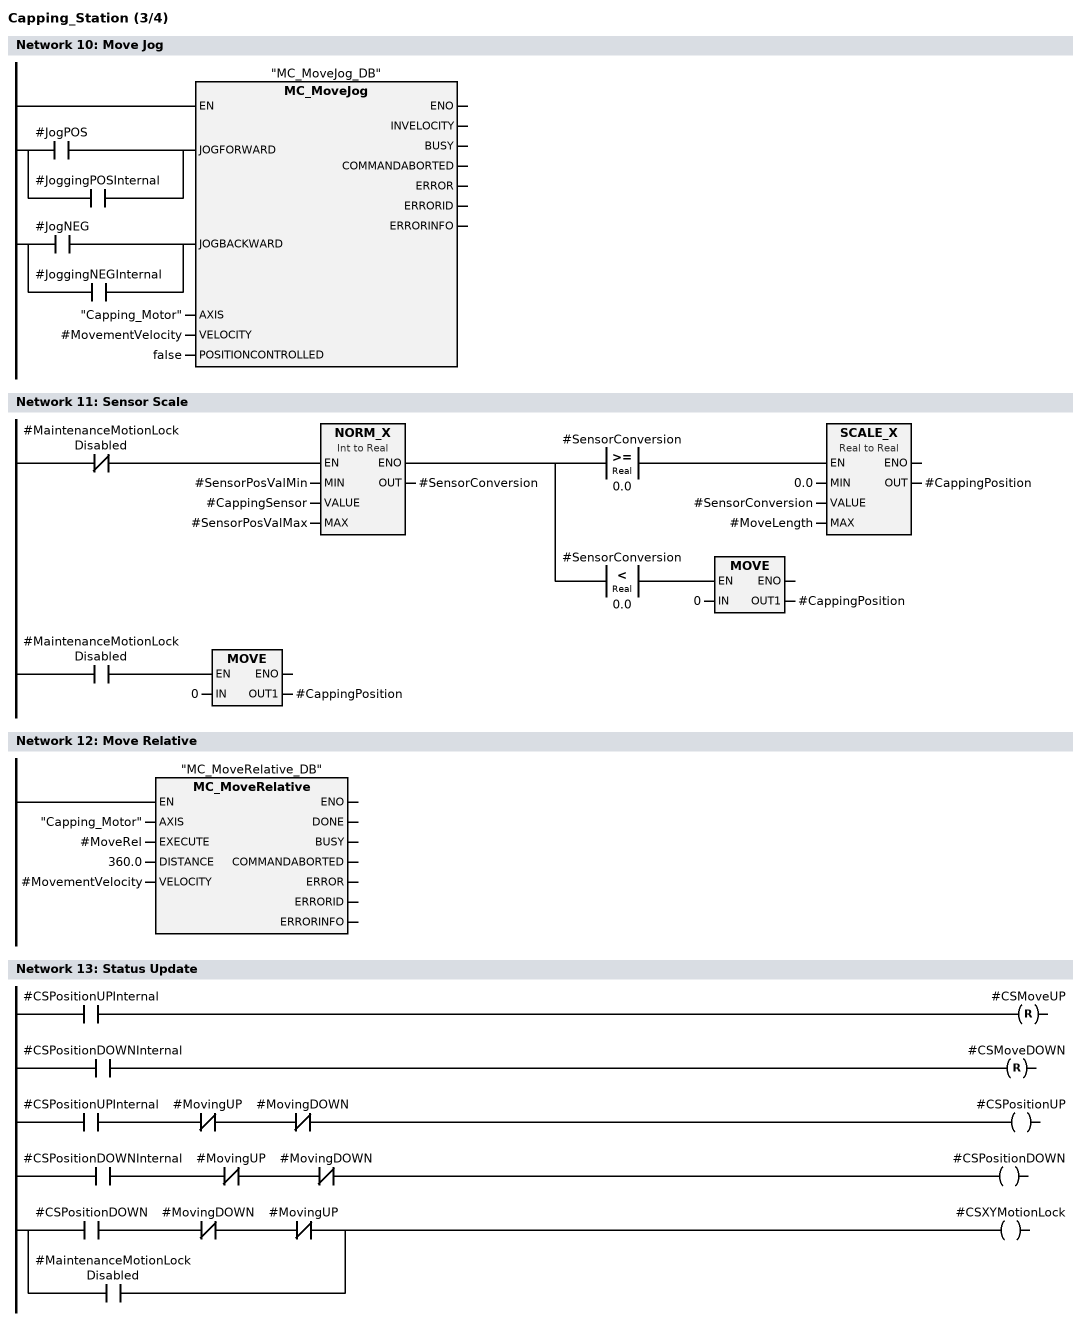
   RUNG wire#powerrail
      "MC_MoveJog_DB".MC_MoveJog(JogForward := wire#w1, JogBackward := wire#w2, Axis := "Capping_Motor", Velocity := #MovementVelocity, PositionControlled := false, InVelocity =>, Busy =>, CommandAborted =>, Error =>, ErrorID =>, ErrorInfo =>)
   END_RUNG
   RUNG wire#powerrail
      Contact( #JogPOS )
   END_RUNG wire#w1
   RUNG wire#powerrail
      Contact( #JoggingPOSInternal )
   END_RUNG wire#w1
   RUNG wire#powerrail
      Contact( #JogNEG )
   END_RUNG wire#w2
   RUNG wire#powerrail
      Contact( #JoggingNEGInternal )
   END_RUNG wire#w2
   // the same network as SCL:
   "MC_MoveJog_DB"(JogForward := #JogPOS OR #JoggingPOSInternal,   // MC_MoveJog
                   JogBackward := #JogNEG OR #JoggingNEGInternal,
                   Axis := "Capping_Motor",
                   Velocity := #MovementVelocity,
                   PositionControlled := false);
END_REGION

REGION Network 11: Sensor Scale
   RUNG wire#powerrail
      I_Contact( #MaintenanceMotionLockDisabled )
      { S7_Templates := "[SrcType := Int, DestType := Real]" } Normalize(min := #SensorPosValMin, value := #CappingSensor, max := #SensorPosValMax, out => #SensorConversion)
      wire#w1
      { S7_Templates := "SrcType := Real" } GE_Contact(in1 := #SensorConversion, in2 := 0.0)
      { S7_Templates := "[SrcType := Real, DestType := Real]" } Scale(min := 0.0, value := #SensorConversion, max := #MoveLength, out => #CappingPosition)
   END_RUNG
   RUNG wire#w1
      { S7_Templates := "SrcType := Real" } LT_Contact(in1 := #SensorConversion, in2 := 0.0)
      Move(in := 0, out1 => #CappingPosition)
   END_RUNG
   RUNG wire#powerrail
      Contact( #MaintenanceMotionLockDisabled )
      Move(in := 0, out1 => #CappingPosition)
   END_RUNG
   // the same network as SCL:
   #_w1 := NOT #MaintenanceMotionLockDisabled;
   IF #_w1 THEN
       #SensorConversion := NORM_X(MIN := #SensorPosValMin, VALUE := #CappingSensor, MAX := #SensorPosValMax);
   END_IF;
   IF #_w1 AND (#SensorConversion >= 0.0) THEN
       #CappingPosition := SCALE_X(MIN := 0.0, VALUE := #SensorConversion, MAX := #MoveLength);
   END_IF;
   IF #_w1 AND (#SensorConversion < 0.0) THEN #CappingPosition := 0; END_IF;
   IF #MaintenanceMotionLockDisabled THEN #CappingPosition := 0; END_IF;
END_REGION

REGION Network 12: Move Relative
   RUNG wire#powerrail
      "MC_MoveRelative_DB".MC_MoveRelative(Axis := "Capping_Motor", Execute := #MoveRel, Distance := 360.0, Velocity := #MovementVelocity, Done =>, Busy =>, CommandAborted =>, Error =>, ErrorID =>, ErrorInfo =>)
   END_RUNG
   // the same network as SCL:
   "MC_MoveRelative_DB"(Axis := "Capping_Motor",   // MC_MoveRelative
                        Execute := #MoveRel,
                        Distance := 360.0,
                        Velocity := #MovementVelocity);
END_REGION

REGION Network 13: Status Update
   RUNG wire#powerrail
      Contact( #CSPositionUPInternal )
      R_Coil( #CSMoveUP )
   END_RUNG
   RUNG wire#powerrail
      Contact( #CSPositionDOWNInternal )
      R_Coil( #CSMoveDOWN )
   END_RUNG
   RUNG wire#powerrail
      Contact( #CSPositionUPInternal )
      I_Contact( #MovingUP )
      I_Contact( #MovingDOWN )
      Coil( #CSPositionUP )
   END_RUNG
   RUNG wire#powerrail
      Contact( #CSPositionDOWNInternal )
      I_Contact( #MovingUP )
      I_Contact( #MovingDOWN )
      Coil( #CSPositionDOWN )
   END_RUNG
   RUNG wire#powerrail
      Contact( #CSPositionDOWN )
      I_Contact( #MovingDOWN )
      I_Contact( #MovingUP )
      wire#w1
      Coil( #CSXYMotionLock )
   END_RUNG
   RUNG wire#powerrail
      Contact( #MaintenanceMotionLockDisabled )
   END_RUNG wire#w1
   // the same network as SCL:
   IF #CSPositionUPInternal THEN #CSMoveUP := FALSE; END_IF;
   IF #CSPositionDOWNInternal THEN #CSMoveDOWN := FALSE; END_IF;
   #CSPositionUP := #CSPositionUPInternal AND NOT #MovingUP AND NOT #MovingDOWN;
   #CSPositionDOWN := #CSPositionDOWNInternal AND NOT #MovingUP AND NOT #MovingDOWN;
   #CSXYMotionLock := (#CSPositionDOWN AND NOT #MovingDOWN AND NOT #MovingUP) OR #MaintenanceMotionLockDisabled;
END_REGION

REGION Network 14: Moves counter
